# B&R Automation Studio project perfxxl (part 9)

#### flowcontrol.c
```c
#ifdef _DEFAULT_INCLUDES
	#include <AsDefault.h>
#endif
/*************************************************************************************************
 Flow control

 - checking Flow control sensor

*************************************************************************************************/

#include "egmglob_var.h"

BOOL				Pulse_1s,Overflow;
TON_10ms_typ		PulseTimer1;

_LOCAL	BOOL		CounterReset;

_LOCAL INT			DevCircFlowInv,PrewashFlowInv,RinseFlowInv,
					GumFlowInv, ReplFlowInv, TopUpFlowInv;

void FlowControl(FlowCount_type *FC,BOOL In, INT MinFreq)
{
	void NoFlow(void)
	{
		FC->LastCV = 0;
		FC->Flowing = FALSE;
		FC->EdgeCounter.RESET = TRUE;

		FC->LitersPerHour = 0;
		FC->LitersPerMinute = 0;
		FC->Frequency = 0;
		FC->OverflowCounter = 0;
	}

	if (Pulse_1s)
	{
		/*
		 * Sonderfall: wenn genau vor einem Zyklus ein Overflow stattfand
		 * dann ist aktueller Zählerstand = letzter Zählerstand = 0
		 * in dem Fall soll kein Reset erfolgen, sondern eine
		 * weitere Sekunde gewartet werden
		 */
		if( !Overflow )
		{
			if(FC->EdgeCounter.CV > FC->LastCV)
			{
				FC->Frequency = (FC->EdgeCounter.CV - FC->LastCV);
				FC->LastCV = FC->EdgeCounter.CV;
				if( FC->Frequency >= MinFreq )
				{
					FC->Flowing = TRUE;
					FC->LitersPerHour = (FC->Frequency / (REAL)FC->PulsesPerLiter)*3600.0;
					FC->LitersPerMinute = (FC->Frequency / (REAL)FC->PulsesPerLiter)*60.0;
				}
				else
					NoFlow();
			}
			else /* counter value has not been increased since 1 sec.: no flow */
				NoFlow();
		} /* if(!Overflow) */
		Overflow = FALSE;
	} /* if(Pulse_1s) */

/* reset value from somewhere else */
	if(FC->ResetMlFlown)
	{
		FC->ResetMlFlown = 0;
		FC->EdgeCounter.RESET = TRUE;
		FC->MlFlown = 0;
		FC->LastCV = 0;
		FC->OverflowCounter = 0;
	}

	if(CounterReset)
	{
		NoFlow();
		FC->MlFlown = 0;
	}

	/* counter overflow at 30000 */
	if(FC->EdgeCounter.CV >= 30000)
	{
		FC->EdgeCounter.RESET = TRUE;
		FC->LastCV = 0;
		FC->OverflowCounter++;
		Overflow = TRUE;
	}
	FC->EdgeCounter.CU = In;
	CTU(&(FC->EdgeCounter));
	FC->EdgeCounter.RESET = FALSE;

	if( FC->EdgeCounter.CV != 0 )
		FC->MlFlown = 1000.0 *
					( ((30000.0 * FC->OverflowCounter) + FC->EdgeCounter.CV)
					    / (REAL)FC->PulsesPerLiter
					 );
}

void InitFlowControl(FlowCount_type *FC)
{
	FC->EdgeCounter.CU = 0;
	FC->EdgeCounter.RESET = 1;
	FC->EdgeCounter.PV = 0;
	FC->OverflowCounter = 0;
	FC->LastCV = 0;
	FC->MlFlown = 0;
	FC->ResetMlFlown = 0;
}

_INIT void init(void)
{
	InitFlowControl(&GumFC);
	InitFlowControl(&ReplFC);
	InitFlowControl(&TopUpFC);

	PulseTimer1.IN = 0;
	PulseTimer1.PT = 100;
}

_CYCLIC void cyclic(void)
{
	DevCircFlowInv = !DevCircFlowInput;
	PrewashFlowInv = !PrewashFlowInput;
	RinseFlowInv = !RinseFlowInput;
	GumFlowInv = !GumFC.Flowing;
	ReplFlowInv = !ReplFC.Flowing;
	TopUpFlowInv = !TopUpFC.Flowing;

	PulseTimer1.IN = 1;
	if(PulseTimer1.Q)
		PulseTimer1.IN = 0;
	TON_10ms(&PulseTimer1);
	Pulse_1s = PulseTimer1.Q;

	if(    (EGMGlobalParam.GumPulsesPerLiter < 500)
		|| (EGMGlobalParam.GumPulsesPerLiter > 5000) )
		EGMGlobalParam.GumPulsesPerLiter = 1200;

	if(    (EGMGlobalParam.ReplenisherPulsesPerLiter < 500)
		|| (EGMGlobalParam.ReplenisherPulsesPerLiter > 5000) )
		EGMGlobalParam.ReplenisherPulsesPerLiter = 1200;

	if(    (EGMGlobalParam.DeveloperPulsesPerLiter < 500)
		|| (EGMGlobalParam.DeveloperPulsesPerLiter > 5000) )
		EGMGlobalParam.DeveloperPulsesPerLiter = 1200;

	GumFC.PulsesPerLiter = EGMGlobalParam.GumPulsesPerLiter;
	ReplFC.PulsesPerLiter = EGMGlobalParam.ReplenisherPulsesPerLiter;
	TopUpFC.PulsesPerLiter = EGMGlobalParam.DeveloperPulsesPerLiter;

	FlowControl(&GumFC,GumFlowInput,2);
	FlowControl(&ReplFC,ReplFlowInput,9);
	FlowControl(&TopUpFC,TopUpFlowInput,9);

}
```

### Program Logical/Processor/lccount (ANSIC, version 0.00.0)

#### lccount.c
```c
#ifdef _DEFAULT_INCLUDES
	#include <AsDefault.h>
#endif
/******************************************************************************************/
/*	LCCount aufrufen (Zeitbasis für Regler)*/
/**/
/******************************************************************************************/

#include "EGMglob_var.h"
#include <loopcont.h>

#define MM_PER_PULSE (251.0/17.0)

R_TRIGtyp	RPMSignalEdgeR;
/*timer für die Messung der Periodendauer des Antriebs-Taktes*/
REAL	tmpval,tmpval2,PeriodTime; /* in sec */

CTUtyp	PlateLengthCounter;

/*timer für die Messung der Periodendauer des Antriebs-Taktes*/
TON_typ	PeriodTimeRPM;
/*timer für die Messung der Verzögerung Plattenvorderkante->nächster Takt*/
TON_10ms_typ	PlateStartToRPMDelay;
/*timer für die Messung der Verzögerung Plattenhinterkante->nächster Takt*/
TON_10ms_typ	PlateEndToRPMDelay;
/*Var zum Speichern der gemessenen Zeiten*/
UDINT	StartDelay,EndDelay;

R_TRIGtyp	InputSensorEdgeR;
F_TRIGtyp	InputSensorEdgeF;
BOOL	 EnablePulseCounter;

_GLOBAL REAL PlateLength;
/* zum Entprellen des Eingangssensors*/
TON_10ms_typ	InputSensorOnDelay;
TOF_10ms_typ	InputSensorOffDelay;
_LOCAL REAL TEST;

/* ohne Mittelwertbildung */
void MeasureCurrentSpeed(void)
{

	RPMSignalEdgeR.CLK = RPMCheck;
	R_TRIG(&RPMSignalEdgeR);
/* steigende Flanke und timer ist gestartet: Zeit nehmen und stoppen*/
	if(RPMSignalEdgeR.Q )
	{
/* 2.02: Messung per Timer statt Zykluszähler */
		PeriodTime = PeriodTimeRPM.ET * 0.001; /* timer Wert 1 ms */
		PeriodTimeRPM.IN = FALSE;
	}
	else
		PeriodTimeRPM.IN = TRUE;
	PeriodTimeRPM.PT = 10000;
/* wenn 10 sec lang kein Takt, dann ist die Periodendauer 0 */
	if(PeriodTimeRPM.Q)
		PeriodTime = 0;

 	TON(&PeriodTimeRPM);
/* ENDE Periodendauer des Taktes messen*/
/*-------------------------------------------------------------------------------------------*/

/*-------------------------------------------------------------------------------------------*/
/* START Geschwindigkeit und Plattenlänge errechnen*/
/* Periodendauer ist gegen 0: Antrieb läuft nicht*/
/* Abfrage wichtig, da durch PeriodTime geteilt wird !!*/
	if (PeriodTime < 0.05)/* kürzer als 50 ms : ungültig, wäre 12 m/min*/
	{
		EGMGlobalParam.CurrentPlateSpeed = 0;
	}
	else
	{
/* 251mm/U / 17Takte/U =14.76 mm/Takt steht in MM_PER_PULSE */
/*PeriodTime*0.01 weil Timerwert in 10ms */
/* *0.06 weil Speed in m/min, Ergebnis vorher ist in mm/s*/
/* gilt so nur, wenn die Speed konstant ist, um schwankungen zu erfassen müsste man integrieren*/

	 	EGMGlobalParam.CurrentPlateSpeed = (MM_PER_PULSE / (PeriodTime))*0.06;
		tmpval = EGMGlobalParam.CurrentPlateSpeed / EGMGlobalParam.MainMotorFactor;
		if (tmpval <= 32767.0)
			EGMMainMotor.RealRpm = (INT)tmpval;
		else
			EGMMainMotor.RealRpm = 32767;

	}
/* ENDE Geschwindigkeit und Plattenlänge errechnen*/
/*-------------------------------------------------------------------------------------------*/
}

void MeasurePlateLength(void)
{

/**********************************************************************************/
/* Plattenlänge ermitteln*/

/*
Strategie für erhöhte Genauigkeit:
	- kontinuierlich Periodendauer des Taktsignals vom Antrieb messen (jede 2. Periode)
	- Zeit vom Erkennen des Plattenanfangs bis zum nächsten Takt messen
	- Zeit vom Erkennen des Plattenendes bis zum nächsten Takt messen
	- aus den gezählten Takten und den gemessenen Zeiten die Plattenlänge
	  ermitteln
*/

/*Entprellen je 1 sec*/
	InputSensorOnDelay.PT = 100;
	InputSensorOffDelay.PT = 100;
	InputSensorOnDelay.IN = InputSensor;
	InputSensorOffDelay.IN = InputSensor;
	TON_10ms(&InputSensorOnDelay);
	TOF_10ms(&InputSensorOffDelay);
	InputSensorEdgeR.CLK = InputSensorOnDelay.Q;
	InputSensorEdgeF.CLK = InputSensorOffDelay.Q;
	R_TRIG(&InputSensorEdgeR);
	F_TRIG(&InputSensorEdgeF);

/*-------------------------------------------------------------------------------------------*/
/* START Messung Verzögerung Plattenvorderkante->nächster Takt*/
/*mit steigender Flanke des Sensors Zeitmessung starten*/
	PlateStartToRPMDelay.PT = 60000;
	if (InputSensorEdgeR.Q && !PlateStartToRPMDelay.IN)
		PlateStartToRPMDelay.IN = 1;
/*bei der nächsten steigenden Flanke des Taktes die Zeit nehmen*/
/* || PlateStartToRPMDelay.Q nur für den Fall, dass der Antrieb steht o.ä.*/
	if (PlateStartToRPMDelay.IN && (RPMSignalEdgeR.Q || PlateStartToRPMDelay.Q ))
	{
		PlateStartToRPMDelay.IN = 0;
		StartDelay = PlateStartToRPMDelay.ET;
	}
	TON_10ms(&PlateStartToRPMDelay);
/* ENDE Messung Verzögerung Plattenvorderkante->nächster Takt*/
/*-------------------------------------------------------------------------------------------*/

/*-------------------------------------------------------------------------------------------*/
/* START Messung Verzögerung Plattenhinterkante->nächster Takt*/
/*mit steigender Flanke des Sensors Zeitmessung starten*/
	PlateEndToRPMDelay.PT = 60000;
	if (InputSensorEdgeF.Q && !PlateEndToRPMDelay.IN)
		PlateEndToRPMDelay.IN = 1;
/*bei der nächsten steigenden Flanke des Taktes die Zeit nehmen*/
/* || PlateEndToRPMDelay.Q nur für den Fall, dass der Antrieb steht o.ä.*/
	if (PlateEndToRPMDelay.IN && (RPMSignalEdgeR.Q || PlateEndToRPMDelay.Q ))
	{
		PlateEndToRPMDelay.IN = 0;
		EndDelay = PlateEndToRPMDelay.ET;
	}
	TON_10ms(&PlateEndToRPMDelay);
/* ENDE Messung Verzögerung Plattenhinterkante->nächster Takt*/
/*-------------------------------------------------------------------------------------------*/

/*-------------------------------------------------------------------------------------------*/
/* START Zählen der Takte, während Platte durchläuft*/
	CTU(&PlateLengthCounter);

/*bei fallender Flanke den Zähler auswerten*/
	if(InputSensorEdgeF.Q)
	{
/* nicht durch 0 teilen... */
		if(PeriodTime < 0.05)
			tmpval2 = PlateLengthCounter.CV;
		else
			tmpval2 = PlateLengthCounter.CV+ ((REAL)StartDelay)/(PeriodTime*100.0) - ((REAL)EndDelay)/(PeriodTime*100.0);
		PlateLength = tmpval2 * MM_PER_PULSE;
		if (PlateLength < 0.0) PlateLength = 0.0;
		if (PlateLength > 3000.0) PlateLength = 0.0;
		EnablePulseCounter = 0;
	}
/* mit Einlaufstart den Pulszähler enablen*/
	if(InputSensorEdgeR.Q)
	{
		EnablePulseCounter = 1;
	}
	if (EnablePulseCounter)
	{
		PlateLengthCounter.CU = RPMCheck;
	}
/*zur Sicherheit den Pulscounter disablen, wenn keine Platte im Einlaufbereich ist*/
	if ( !InputSensorOnDelay.Q && !InputSensorOffDelay.Q)
		EnablePulseCounter = 0;

/*bei Start einer Platte Zähler resetten, Takte zählen*/
	PlateLengthCounter.RESET = InputSensorEdgeR.Q;

/* ENDE Zählen der Takte, während Platte durchläuft*/
/*-------------------------------------------------------------------------------------------*/
}

_INIT void init(void)
{
	PlateLength = 0;
/*	PeriodTimeCounter = 0;*/
	PeriodTime = 0;
	PeriodTimeRPM.IN = FALSE;
}

_CYCLIC void cyk(void)
{
	LCCounter(&LCCountVar);
	MeasureCurrentSpeed();
	MeasurePlateLength();
}
```

- egmglob_var.h (reference to Logical/GlobalIncludes/egmglob_var.h)

### Program Logical/Processor/egmio (ANSIC, version 0.00.0)

#### egm_in_out.c
```c
#ifdef _DEFAULT_INCLUDES
	#include <AsDefault.h>
#endif
#include "glob_var.h"
#include "egmglob_var.h"

#define OUTMODULES (3)
#define OUTPUTSPERMODULE (12)

_LOCAL    BOOL                EGMModule1Out[12];
_LOCAL    BOOL                EGMModule2Out[12];
_LOCAL    BOOL                EGMModule3Out[12];
_LOCAL    BOOL                EGMModule1In[12];
_LOCAL    BOOL                EGMModule2In[12];

static BOOL dummy;

_INIT void i(void)
{
	MachineType = BLUEFIN_LOWCHEM;
/*	MachineType = BLUEFIN_XS;*/
}

_CYCLIC void c(void)
{

/*
Maschinenlänge in m
	Standard Bluefin 2.80
	XS Bluefin		 2.70
	LowChem Bluefin  2.05
 */

	if(MachineType == BLUEFIN_XS)
	{
		MACHINELENGTH = 2.70;
	/* XS Output */
		EGMModule1Out[0] = Horn;
		EGMModule1Out[1] = LightGreen;
		EGMModule1Out[2] = LightYellow;
		EGMModule1Out[3] = LightRed;
		EGMModule1Out[4] = EGMMainMotor.Enable;
		EGMModule1Out[5] = EGMBrushMotor.Enable;
		EGMModule1Out[6] = Ready;
		EGMModule1Out[7] = NoError;
		EGMModule1Out[8] = ActivateControlVoltage;
		EGMModule1Out[9] = EGMPrewash.Valve;
		EGMModule1Out[10] = EGMRinse.Valve;
		EGMModule1Out[11] = EGMGum.RinseValve;

		EGMModule2Out[0] = HeatingON[0];
		EGMModule2Out[1] = HeatingON[1];
		EGMModule2Out[2] = HeatingON[2];
		EGMModule2Out[3] = HeatingON[3];
		EGMModule2Out[4] = EGMDeveloperTank.HeatingOn;
		EGMModule2Out[5] = EGMGum.Valve;
		EGMModule2Out[6] = EGMDeveloperTank.CoolingOn;
		EGMModule2Out[7] = FALSE;
		EGMModule2Out[8] = FALSE;
		EGMModule2Out[9] = FALSE;
		EGMModule2Out[10] = FALSE;
		EGMModule2Out[11] = FALSE;

		EGMModule3Out[0] = EGMPrewash.Pump;
		EGMModule3Out[1] = EGMRinse.Pump;
		EGMModule3Out[2] = EGMPreheat.FansOn;
		EGMModule3Out[3] = Drying;
		if(EGMGlobalParam.PROV_KitInstalled)
			EGMModule3Out[4] = Out_DevCanister_Circulation;
		else
			EGMModule3Out[4] = EGMDeveloperTank.RegenerationPump;
		EGMModule3Out[5] = EGMGum.Pump;
		EGMModule3Out[6] = EGMDeveloperTank.CirculationPump;
		if(EGMGlobalParam.PROV_KitInstalled)
			EGMModule3Out[7] = Out_DevCanister_Replenish;
		else
			EGMModule3Out[7] = EGMDeveloperTank.Refill;
		EGMModule3Out[8] = FALSE;
		EGMModule3Out[9] = FALSE;
		EGMModule3Out[10] = FALSE;
		EGMModule3Out[11] = FALSE;

	/* XS Input */
		ControlVoltageOk 			= EGMModule1In[0];
		RPMCheck 					= EGMModule1In[1];
		InputSensor 				= EGMModule1In[2];
		EGMPrewash.TankFull 		= EGMModule1In[3];
		EGMRinse.TankFull 			= EGMModule1In[4];
		EGMGum.TankFull				= EGMModule1In[5];
		EGMDeveloperTank.TankFull	= EGMModule1In[6];
/*                                                 7 s.u.ProV */
		OutputSensor				= EGMModule1In[8];
		ServiceKey					= EGMModule1In[9];
		VCP_OK						= EGMModule1In[10];
		if(EGMGlobalParam.PROV_KitInstalled)
		{
			In_DevCanister_Full			= EGMModule1In[7];
			In_DevCanister_Empty		= EGMModule1In[11];
		}
		else
		{
			dummy						= EGMModule1In[7];
			dummy						= EGMModule1In[11];
		}

		GumFlowInput	 			= EGMModule2In[0];
		ReplFlowInput	 			= EGMModule2In[1];
		TopUpFlowInput	 			= EGMModule2In[2];
		DevCircFlowInput 			= EGMModule2In[3];
		PrewashFlowInput	 		= EGMModule2In[4];
		RinseFlowInput	 			= EGMModule2In[5];
/*		In_WasteTankNearlyFull		= EGMModule2In[6];
		In_WasteTankFull 			= EGMModule2In[7];*/
		dummy						= EGMModule2In[8];
		dummy						= EGMModule2In[9];
		dummy						= EGMModule2In[10];
		dummy						= EGMModule2In[11];
	}
	else
	if(MachineType == BLUEFIN_LOWCHEM)
	{
		EGMGlobalParam.PROV_KitInstalled = FALSE;
		MACHINELENGTH = 2.05;
	/* LowChem Output */
		EGMModule1Out[0] = Horn;
		EGMModule1Out[1] = LightGreen;
		EGMModule1Out[2] = LightYellow;
		EGMModule1Out[3] = LightRed;
		EGMModule1Out[4] = EGMMainMotor.Enable;
		EGMModule1Out[5] = EGMBrushMotor.Enable;
		EGMModule1Out[6] = ActivateControlVoltage;
		EGMModule1Out[7] = FALSE;
		EGMModule1Out[8] = FALSE;
		EGMModule1Out[9] = FALSE;
		EGMModule1Out[10] = EGMGum.Valve;
		EGMModule1Out[11] = EGMGum.RinseValve;

		EGMModule2Out[0] = HeatingON[0];
		EGMModule2Out[1] = HeatingON[1];
		EGMModule2Out[2] = EGMDeveloperTank.HeatingOn;
		EGMModule2Out[3] = FALSE;
		EGMModule2Out[4] = FALSE;
		EGMModule2Out[5] = FALSE;
		EGMModule2Out[6] = EGMDeveloperTank.CoolingOn;
		EGMModule2Out[7] = FALSE;
		EGMModule2Out[8] = FALSE;
		EGMModule2Out[9] = FALSE;
		EGMModule2Out[10] = FALSE;
		EGMModule2Out[11] = FALSE;

		EGMModule3Out[0] = EGMPrewash.Pump;
		EGMModule3Out[1] = EGMRinse.Pump;
		EGMModule3Out[2] = EGMPreheat.FansOn;
		EGMModule3Out[3] = Drying;
		EGMModule3Out[4] = EGMDeveloperTank.RegenerationPump;
		EGMModule3Out[5] = EGMGum.Pump;
		EGMModule3Out[6] = EGMDeveloperTank.CirculationPump;
		EGMModule3Out[7] = EGMDeveloperTank.Refill;
		EGMModule3Out[8] = FALSE;
		EGMModule3Out[9] = FALSE;
		EGMModule3Out[10] = Ready;
		EGMModule3Out[11] = NoError;

	/* LowChem Input */
		ControlVoltageOk 			= EGMModule1In[0];
		RPMCheck 					= EGMModule1In[1];
		InputSensor 				= EGMModule1In[2];
		DevCircFlowInput	 		= EGMModule1In[3];
		TopUpFlowInput	 			= EGMModule1In[4];
		EGMGum.TankFull				= EGMModule1In[5];
		EGMDeveloperTank.TankFull	= EGMModule1In[6];
		GumFlowInput				= EGMModule1In[7];
		OutputSensor				= EGMModule1In[8];
		ServiceKey					= EGMModule1In[9];
		VCP_OK						= EGMModule1In[10];
		dummy						= EGMModule1In[11];

		dummy						= EGMModule2In[0];
		ReplFlowInput	 			= EGMModule2In[1];
		dummy						= EGMModule2In[2];
		dummy						= EGMModule2In[3];
		dummy						= EGMModule2In[4];
		dummy						= EGMModule2In[5];
		dummy						= EGMModule2In[6];
		dummy						= EGMModule2In[7];
		dummy						= EGMModule2In[8];
		dummy						= EGMModule2In[9];
		dummy						= EGMModule2In[10];
		dummy						= EGMModule2In[11];
	}
}
```

- egmglob_var.h (reference to Logical/GlobalIncludes/egmglob_var.h)

### Program Logical/Processor/motors (ANSIC, version 0.00.0)

#### motors.c
```c
#ifdef _DEFAULT_INCLUDES
	#include <AsDefault.h>
#endif
/*************************************************************************************************
 Handling of Motors
 - Main Motor (Propulsion of plate)
 - Brush Motor

*************************************************************************************************/

#include "glob_var.h"
#include "egmglob_var.h"
#include <math.h>

TP_10ms_typ		RPMCheckTimer;
F_TRIGtyp 			RPMCheckEdge;
CTUtyp	RPMEdgeCounter;
_LOCAL	UINT	CounterValue;
TON_10ms_typ		BrushMotorOnTimer1,BrushMotorOnTimer2;
TON_10ms_typ		RPMSignalCheckTimer,RPMDeviationTimer;
/* Input delay timer for ControlVoltage signal */
TON_10ms_typ		ControlVoltageOkDelay;

REAL	tmpval;

TON_10ms_typ	PulseTimer1;
BOOL	Pulse_1s;
_LOCAL REAL MainMotorFactorFeet;

_INIT void init()
{
	CounterValue = 0;
	EGMMainMotor.RatedRpm = 0;
	EGMMainMotor.RealRpm = 0;
	EGMMainMotor.Auto = 0;
	EGMMainMotor.Enable = 0;

	EGMBrushMotor.RatedRpm = 0;
	EGMBrushMotor.RealRpm = 0;
	EGMBrushMotor.Auto = 0;
	EGMBrushMotor.Enable = 0;

	BrushMotorOnTimer1.IN = 0;
	BrushMotorOnTimer2.IN = 0;

	PulseTimer1.IN = 0;
	PulseTimer1.PT = 100; /* 1 sec */

}

_CYCLIC void cyclic()
{
	PulseTimer1.IN = 1;
	if(PulseTimer1.Q)
		PulseTimer1.IN = 0;
	TON_10ms(&PulseTimer1);
	Pulse_1s = PulseTimer1.Q;

/* Skalierungsfaktor muss in VC Einheitengruppe "Vorschub" identisch sein !! */
/*	EGMGlobalParam.MainMotorFactor = 9.30814539017914E-05;*/
	MainMotorFactorFeet = EGMGlobalParam.MainMotorFactor / 0.3048;
/* das gleiche für Bürstenmotor */
/*  "Alter" Motortyp*/
/*	EGMGlobalParam.BrushFactor = 180.0/32767.0;*/
/*  "Neuer" Motortyp Siemens*/
/*	EGMGlobalParam.BrushFactor = 230.0/32767.0;*/

/* safety:
 * 	Not a number or out of reasonable range ->set default*/
	if( isnan(EGMGlobalParam.BrushFactor)
	 || (EGMGlobalParam.BrushFactor > 0.02)  /* > ca 655 rpm */
	 || (EGMGlobalParam.BrushFactor < 0.001) /* < ca 32.7 rpm */
	  )
		EGMGlobalParam.BrushFactor = 230.0/32767.0;

/*Main Motor*/
/* safety:
 * 	Not a number or out of reasonable range ->set default*/
	if( isnan(EGMGlobalParam.MainMotorFactor)
	 || (EGMGlobalParam.MainMotorFactor > (10.0/32767.0))
	 || (EGMGlobalParam.MainMotorFactor < 1.0/32767.0)
	  )
		EGMGlobalParam.MainMotorFactor = 3.0/32767.0;

	EGMMainMotor.Manual = !EGMMainMotor.Auto;

/**
Prüfen, ob überhaupt Signale vom Taktsensor kommen:
Wenn Sollwert > 0,2 m/min, dann muss der Countervalue > 0 sein
*/
	RPMSignalCheckTimer.IN = ((CounterValue == 0) && ((EGMMainMotor.RatedRpm * EGMGlobalParam.MainMotorFactor)> 0.2 ));
	RPMSignalCheckTimer.PT = 1000; /* 10 sec */
	TON_10ms(&RPMSignalCheckTimer);
	EGM_AlarmBitField[1] = RPMSignalCheckTimer.Q;

	RPMDeviationTimer.PT = 1000;
	RPMDeviationTimer.IN = ((fabs((EGMGlobalParam.MainMotorFactor*EGMMainMotor.RatedRpm) - EGMGlobalParam.CurrentPlateSpeed)) > 0.5)
							&& !EGM_AlarmBitField[1] && EGMMainMotor.Enable && !CurrentState==S_OFF && ControlVoltageOk;
	TON_10ms(&RPMDeviationTimer);
	EGM_AlarmBitField[27] = RPMDeviationTimer.Q;

/* Messung der Speed über Taktgeber*/
	RPMEdgeCounter.CU = RPMCheck;
	RPMEdgeCounter.PV = 32000; /*soll nicht erreicht werden*/

	CTU(&RPMEdgeCounter);
	RPMEdgeCounter.RESET = 0;

	TP_10ms(&RPMCheckTimer);

	RPMCheckTimer.IN = Pulse_1s;
	RPMCheckTimer.PT = 1000; /*10 sec Messen*/

/*fallende Flanke des Pulstimers auswerten*/
	RPMCheckEdge.CLK	= RPMCheckTimer.Q;
	F_TRIG(&RPMCheckEdge);

	if (RPMCheckEdge.Q)
	{
		CounterValue = RPMEdgeCounter.CV;
		RPMEdgeCounter.RESET = 1;
	}

/*im Automatik-Modus die Auto-Drehzahl übernehmen*/
/*-> im Hand Modus kann man dann die RatedRpm direkt verändern*/
/*Spannung muß schon 5 sec lang anliegen, sonst erkennt FU das Signal nicht zuverlässig*/
	ControlVoltageOkDelay.IN = ControlVoltageOk;
	ControlVoltageOkDelay.PT = 500;
	TON_10ms(&ControlVoltageOkDelay);
	if (EGMMainMotor.Auto && ControlVoltageOkDelay.Q)
	{
		EGMMainMotor.Enable = 1;	/* Freigabe Ausgang an FU */
		EGMMainMotor.RatedRpm = EGMMainMotor.AutoRatedRpm;	/* Drehzahl Ausgang an FU */
	}

	if (!ControlVoltageOk)
	{
		EGMMainMotor.Enable = 0;	/* Freigabe Ausgang an FU */
		EGMMainMotor.Auto = 0;
	}

/*************************************************************************************************/

/*Brush Motor*/
	EGMBrushMotor.Manual = !EGMBrushMotor.Auto;
/*keine Messung: Ist = Soll*/
	EGMBrushMotor.RealRpm = EGMBrushMotor.RatedRpm;
/*im Automatik-Modus die Auto-Drehzahl übernehmen*/
/*-> im Hand Modus kann man dann die RatedRpm direkt verändern*/
	if (EGMBrushMotor.Auto && ControlVoltageOkDelay.Q)
	{
		EGMBrushMotor.Enable = 1;	/* Freigabe Ausgang an FU */
/*
		if (BrushMotorOnTimer2.IN )
			EGMBrushMotor.RatedRpm = 150.0 / EGMGlobalParam.BrushFactor;
		else
 */
			EGMBrushMotor.RatedRpm = EGMBrushMotor.AutoRatedRpm;	/* Drehzahl Ausgang an FU */
	}

	if (!ControlVoltageOk)
	{
		EGMBrushMotor.Enable = 0;	/* Freigabe Ausgang an FU */
		EGMBrushMotor.Auto = 0;
	}

	if (EGMBrushMotor.Auto && (EGMBrushMotor.RatedRpm < 100.0/EGMGlobalParam.BrushFactor) )
	{
		BrushMotorOnTimer1.IN = 1;
	}
	else
		BrushMotorOnTimer1.IN = 0;

	BrushMotorOnTimer1.PT = 9000; /* alle 1,5 min*/
	TON_10ms(&BrushMotorOnTimer1);

	BrushMotorOnTimer2.PT = 2000; /* 20 sec*/
	TON_10ms(&BrushMotorOnTimer2);

/* nach Zeit die Bürsten hochdrehen*/
	if (BrushMotorOnTimer1.Q  )
	{
		BrushMotorOnTimer2.IN = 1;
	}

	if (BrushMotorOnTimer2.Q)
	{
		BrushMotorOnTimer2.IN = 0;
	}
}
```

### Program Logical/Processor/preheat (ANSIC, version 0.00.0)

#### preheat.c
```c
#ifdef _DEFAULT_INCLUDES
	#include <AsDefault.h>
#endif
/*************************************************************************************************
 Handling of Preheat

 - Heating, Temperature Measurement

*************************************************************************************************/

#include "EGMglob_var.h"

extern void PreheatPID(void);
extern void PreheatPID_DefaultParam(void);

int i;
_GLOBAL BOOL	HeatingON[4];
_INIT void init()
{

	PreheatPID_DefaultParam();
}

_CYCLIC void cyclic()
{

	PreheatPID();
	return;
}
```

#### preheat_pid.c
```c
#ifdef _DEFAULT_INCLUDES
	#include <AsDefault.h>
#endif
/*****************************************************************************************/
/*	Preheat regelung mit LoopCont Library*/
/*	wird aus EGMPreheat.c aufgerufen*/
/*****************************************************************************************/

/*
#define TESTCURVE
*/
/**/
#undef TESTCURVE
/**/

#include <math.h>
#include "EGMglob_var.h"
#include "auxfunc.h"

/*für Sollwertnachführung*/
#define NUMBER_OF_POINTS		720 /*2h lang alle 10 sec ein wert*/
#define NUMBER_OF_SECONDS	7200 /*2h */
/*für Stabilitätscheck*/
#define NUMBER_OF_RANGECHECK_SECONDS	30
#define OVERHEATTEMP 500	/* 50 °C über der Solltemp.*/

_GLOBAL SINT IOConfiguration	_VAR_RETAIN;

_LOCAL	LCPWM_DMod_typ		LCPWM_DMod_var[MAX_NUMBER_OF_CONTROLLERS];
_LOCAL	LCPIDpara_typ			LCPIDpara_var[MAX_NUMBER_OF_CONTROLLERS];
_LOCAL	LCPID_typ				LCPID_var[MAX_NUMBER_OF_CONTROLLERS];
_LOCAL	LCPIDAutoTune_typ		LCPIDAutoTune_var[MAX_NUMBER_OF_CONTROLLERS];
_LOCAL	LCCurveByPoints_typ	LCCurveByPoints_var,LCCurveByPoints_var2;

/*Feld für Kurve der Sollwertnachführung*/
/* e-Funktion*/
_LOCAL lcCurveByPoints_TabEntry_type   CurveByPoints_Table[NUMBER_OF_POINTS];
/* Korrekturen der e-Funktion*/
_LOCAL lcCurveByPoints_TabEntry_type   CurveByPoints_Table2[15];

_LOCAL	BOOL 	StartAutoTune;
_LOCAL	BOOL	TriggerLogging,TriggerLoggingOld;
TON_10ms_typ	Pulse,PulseTimer1;
TON_10ms_typ		HeatingFailureTimer[MAX_NUMBER_OF_CONTROLLERS];

int i;
_GLOBAL int	Values[350];
_GLOBAL int	AmbientValues[350];

int	RangeCheckArray[MAX_NUMBER_OF_CONTROLLERS][NUMBER_OF_RANGECHECK_SECONDS];
int ValueCount,RangeCheckCount,SPTrackCount;
BOOL flag[MAX_NUMBER_OF_CONTROLLERS];
_GLOBAL BOOL RedrawCurve,PreheatParamEnter;
_GLOBAL	UINT	SamplingTime;
BOOL	StopSPTracking;
BOOL	Overheated;
INT LastTemp[MAX_NUMBER_OF_CONTROLLERS];

R_TRIGtyp	InputSensorEdgeR;
F_TRIGtyp	InputSensorEdgeF;
TON_10ms_typ	InputSensorOnDelay;
TOF_10ms_typ	InputSensorOffDelay;
int	PlateInputCounter;
int TempCorrectionValue;
int SecWithoutPlate;

/* depending on Bluefin-Variant: Standard or 1250 */
_LOCAL    INT                 ActualNumberOfControllers;

void Preset_CorrCurve(void)
{
	int i;
	REAL k;

/*e-Funktion für Startup erzeugen*/
	for (i=0;i<NUMBER_OF_POINTS;i++)
	{
		CurveByPoints_Table[i].x = i*(NUMBER_OF_SECONDS / NUMBER_OF_POINTS) ;

		k = -((float)NUMBER_OF_SECONDS / (float) NUMBER_OF_POINTS)  / (60.0* EGMPreheatParam.SetPointCorrTMin);
		CurveByPoints_Table[i].y = EGMPreheatParam.SetPointCorrMax * exp(k*i);
	}

/*initialisieren der Korrekturkurve für die e-Funktion*/
	for (i=0;i<15;i++)
	{
		CurveByPoints_Table2[i].x = 0;
		CurveByPoints_Table2[i].y = 0;
	}
/*und mit Stützpunkten füllen*/
/* 1 */
	CurveByPoints_Table2[0].x = 0;
	CurveByPoints_Table2[0].y = 0;
/* 2 */
	CurveByPoints_Table2[1].x = 180;
	CurveByPoints_Table2[1].y = -50;
/* 3 */
	CurveByPoints_Table2[2].x = 300;
	CurveByPoints_Table2[2].y = -80;
/* 4 */
	CurveByPoints_Table2[3].x = 540;
	CurveByPoints_Table2[3].y = -90;
/* 5 */
	CurveByPoints_Table2[4].x = 840;
	CurveByPoints_Table2[4].y = -110;
/* 6 */
	CurveByPoints_Table2[5].x = 1200;
	CurveByPoints_Table2[5].y = -80;
/* 7 */
	CurveByPoints_Table2[6].x = 1740;
	CurveByPoints_Table2[6].y = -60;
/* 8 */
	CurveByPoints_Table2[7].x = 2700;
	CurveByPoints_Table2[7].y = -30;
/* 9 */
	CurveByPoints_Table2[8].x = 3480;
	CurveByPoints_Table2[8].y = -10;
/* 10 */
	CurveByPoints_Table2[9].x = 3660;
	CurveByPoints_Table2[9].y = 0;
/* 11 */
	CurveByPoints_Table2[10].x = 4860;
	CurveByPoints_Table2[10].y = 0;
/* 12 */
	CurveByPoints_Table2[11].x = 5400;
	CurveByPoints_Table2[11].y = 10;
/* 13 */
	CurveByPoints_Table2[12].x = 6000;
	CurveByPoints_Table2[12].y = 25;
/* 14 */
	CurveByPoints_Table2[13].x = 6660;
	CurveByPoints_Table2[13].y = 19;

}

void PreheatPID_DefaultParam(void)
{
	int j;

/* depending on IO config we have 2 or 4 Controllers running*/
	switch (IOConfiguration)
	{
		case 1 /* Standard Bluefin */:
		{
			ActualNumberOfControllers = 2;
			break;
		}
		case 2 /* Bluefin 1250 */:
		{
			ActualNumberOfControllers = 4;
			break;
		}
		default:
		{
			ActualNumberOfControllers = 2;
			break;
		}
	}
	PreheatParamEnter = 0;
	StopSPTracking = 0;
	SamplingTime = 100;
	SPTrackCount = 0;
	PulseTimer1.PT = 100;

	LCCurveByPoints_var.ptr_table = &CurveByPoints_Table[0];
	LCCurveByPoints_var.NoOfPoints = NUMBER_OF_POINTS;

	LCCurveByPoints_var2.ptr_table = &CurveByPoints_Table2[0];
	LCCurveByPoints_var2.NoOfPoints = 14;

	Preset_CorrCurve();

	for (i=0;i<ActualNumberOfControllers;i++)
	{
		LCPWM_DMod_var[i].tminpuls			= 10;  /* 10 ms kürzester Puls bzw pause*/
		LCPWM_DMod_var[i].tperiod			= 200;  /*Periodendauer 0,2 sec*/
		LCPWM_DMod_var[i].enable			= 1;
		LCPWM_DMod_var[i].max_value	= 100;
		LCPWM_DMod_var[i].min_value		= 0;

/*Sollwertabschwächung (1=AUS)*/
		LCPIDpara_var[i].Kw						= 1;
/*windup Dämpfung: 0=AUS*/
		LCPIDpara_var[i].Kfbk						= 0;
		LCPIDpara_var[i].enable					= 1;
		LCPIDpara_var[i].Y_max				= 100;
		LCPIDpara_var[i].Y_min					= 0;
		LCPIDpara_var[i].dY_max				= 0; /* 0= keine Rampe*/
	/*
	Rückführmodus der Stellgröße
	LCPID_FBK_MODE_INTERN: intern
	LCPID_FBK_MODE_EXTERN: extern für Ablöseregelung
	LCPID_FBK_MODE_EXT_SELECTOR: extern für Selektorregelung. In diesem Modus wird der I-Anteil des momentan nicht selektierten Reglers (Y_fbk ? Y) nach der
	Formel Yi = Y_fbk – Yp – Yd – A dem Eingang Y_fbk nachgeführt.
	*/
		LCPIDpara_var[i].fbk_mode				= LCPID_FBK_MODE_INTERN;
	/*
	Differenziermodus
	LCPID_D_MODE_X: nur -X (Istwert)
	LCPID_D_MODE_E: e (Regelabweichung, wie bei einem Standard- PID- Regler )
	*/
		LCPIDpara_var[i].d_mode				= LCPID_D_MODE_X;
	/*
	Rechenmodus:
	LCPID_CALC_MODE_EXACT: Genau (Alle Berechnungen erfolgen in Double Float - keine Rundungsfehler, auf SG3-Zentraleinheiten lange Rechenzeiten).
	LCPID_CALC_MODE_FAST: Schnell (Alle Berechnungen erfolgen in Integer - es kann zu geringfügigen Rundungsfehlern kommen, wird auch auf SG3-Zentraleinheiten sehr schnell gerechnet)
	*/
		LCPIDpara_var[i].calc_mode			= LCPID_CALC_MODE_EXACT;

/* Reglerbaustein LCPID*/
		LCPID_var[i].enable					= 1;
/*Stellgröße Handbetrieb */
		LCPID_var[i].Y_man					= 0;
	/*Aufschaltgröße*/
		LCPID_var[i].A							= 0;
	/*I-Anteil einfrieren*/
		LCPID_var[i].hold_I					= 0;

/* Autotune*/
		LCPIDAutoTune_var[i].enable				= 1;
		LCPIDAutoTune_var[i].Y_max				= 100;
		LCPIDAutoTune_var[i].Y_min				= 0;
		LCPIDAutoTune_var[i].P_manualAdjust		= 0;
		LCPIDAutoTune_var[i].I_manualAdjust		= 0;
		LCPIDAutoTune_var[i].D_manualAdjust		= 0;

		EGMPreheat.Auto[i] = 0;

		TriggerLogging = 0;
		for(j=0;j<NUMBER_OF_RANGECHECK_SECONDS;j++)
			RangeCheckArray[i][j] = 200;
	}
	RangeCheckCount = 0;
	i=0;
	ValueCount = 0;
	InputSensorOnDelay.IN = 0;
	InputSensorOffDelay.IN = 0;
	SecWithoutPlate = 0;
	TempCorrectionValue = 0;
	for(i=0;i<ActualNumberOfControllers;i++)
	{
		LastTemp[i] = 0;
		HeatingFailureTimer[i].IN = 0;
		HeatingFailureTimer[i].PT = 1000;
	}
}

/***********************************************************************
*                                                                      *
*                                                                      *
*     Sollwert pro Platte sukzessive erhöhen, nach Zeit ohne Platte    *
*     wieder verringern                                                *
*                                                                      *
*                                                                      *
***********************************************************************/
void SetpointCorrectionPerPlate(void)
{
/*Flankenerkennung Inputsensor */
	InputSensorEdgeR.CLK = InputSensorOnDelay.Q;
	InputSensorEdgeF.CLK = InputSensorOffDelay.Q;
	R_TRIG(&InputSensorEdgeR);
	F_TRIG(&InputSensorEdgeF);

	InputSensorOnDelay.PT = 100;
	InputSensorOffDelay.PT = 100;
/*Entprellen je 1 sec*/
	InputSensorOnDelay.IN = InputSensor;
	InputSensorOffDelay.IN = InputSensor;
	TON_10ms(&InputSensorOnDelay);
	TOF_10ms(&InputSensorOffDelay);

	if( InputSensor )
		SecWithoutPlate = 0;
	else
	if( PulseTimer1.Q ) /* Pulse every sec */
	{
		SecWithoutPlate++;
		if( (SecWithoutPlate % 60) == 0) /* every minute */
		{
			TempCorrectionValue += EGMPreheatParam.IncPerMinute;
			if( TempCorrectionValue > 0 )
				TempCorrectionValue = 0;
		}
	}

/* Platte läuft ein */
	if( InputSensorEdgeF.Q )
	{
		SecWithoutPlate = 0;	/* nur zur Sicherheit */
/* wenn Umgebunstemp. > Schwellwert*/
		if( EGMPreheat.AmbientTemp[0] > EGMPreheatParam.AmbientThreshold )
		{
			TempCorrectionValue -= EGMPreheatParam.DecPerPlate;
			if( abs(TempCorrectionValue) > abs(EGMPreheatParam.MaxInc) )
				TempCorrectionValue = EGMPreheatParam.MaxInc;
		}
	}

}

/***********************************************************************
*                                                                      *
*     PID Regler Funktionalität für beide Preheat Kreise               *
*                                                                      *
*                                                                      *
***********************************************************************/
void PreheatPID(void)
{
	int j;
	int k;
/*
	SetpointCorrectionPerPlate();
*/
	TempCorrectionValue = 0; /* rausnehmen, wenn Aufruf von SetpointCorrectionPerPlate
	                          * wieder einkommentiert wird !!
                              */

/* depending on IO config we have 2 or 4 Controllers running*/
	switch (IOConfiguration)
	{
		case 1 /* Standard Bluefin */:
		{
			ActualNumberOfControllers = 2;
			break;
		}
		case 2 /* Bluefin 1250 */:
		{
			ActualNumberOfControllers = 4;
			break;
		}
		default:
		{
			ActualNumberOfControllers = 2;
			break;
		}
	}

	for (j=0;j<ActualNumberOfControllers;j++)
		EGMPreheat.HeatingOn[j] = HeatingON[j];

/* Preheat enabled: Fans on as soon as Controlvoltage is on*/
	if( EGMPreheat.Enable )
		EGMPreheat.FansOn = ControlVoltageOk;
	else /* Preheat Off and Temp. in both Heatings < 100 °C
	      * or Emergency stop
	      * -> Fans OFF
	      */
	if( !ControlVoltageOk ||
	    (EGMPreheat.RealTemp[0] < 1000
	 &&  EGMPreheat.RealTemp[1] < 1000
	 && (LCPWM_DMod_var[0].x == 0)
	 && (LCPWM_DMod_var[1].x == 0))
	  )
		EGMPreheat.FansOn = 0;
	else	/* Preheat OFF, Controlvoltage ON, but both heatings >110 °C
	         * or one heating is ON -> Fans on
	         */
	if( ((EGMPreheat.RealTemp[0] > 1100) && ( EGMPreheat.RealTemp[1] > 1100 ))
	   || (LCPWM_DMod_var[0].x != 0)
	   || (LCPWM_DMod_var[1].x != 0)
	)
		EGMPreheat.FansOn = 1;

/**
Heizung defekt erkennen:
Ausgang 100% aber Temperatur steigt nicht
Erkennung für beide Heizkreise einzeln
**/
	for (i = 0;i<ActualNumberOfControllers;i++)
	{
		HeatingFailureTimer[i].IN = (LCPWM_DMod_var[i].x == 100) && !HeatingFailureTimer[i].Q;
		TON_10ms(&HeatingFailureTimer[i]);

		if( HeatingFailureTimer[i].Q )
		{
			/*
			 * 10 sec 100% Heating, but no rising temp. -> Alarm on
			*/
/* alarms for 1 and 2 are number 19 and 20*/
			if(i<2)
			{
				if( EGMPreheat.RealTemp[i] <= LastTemp[i]+10)
					EGM_AlarmBitField[19+i] = 1;
				else	/* Temp. did rise: Alarm off*/
					EGM_AlarmBitField[19+i] = 0;
			}
/* alarms for 3 and 4 are number 29 and 30*/
			else
			{
				if( EGMPreheat.RealTemp[i] <= LastTemp[i]+10)
					EGM_AlarmBitField[29+i] = 1;
				else	/* Temp. did rise: Alarm off*/
					EGM_AlarmBitField[29+i] = 0;
			}

			/* save current temp. for next check in 10 sec */
			LastTemp[i] = EGMPreheat.RealTemp[i];
		}
/* Heating off, or controller doesn't heat 100% -> Alarm Off*/
		if (LCPWM_DMod_var[i].x < 100)
		{
			if(i<2)
				EGM_AlarmBitField[19+i] = 0;
			else
				EGM_AlarmBitField[29+i] = 0;
		}
	}

/*Sampling der Werte für die Kurve mit einstellbarer Samplingzeit*/
	if (SamplingTime<10) SamplingTime = 100;
	Pulse.PT = SamplingTime;
	TON_10ms(&Pulse);
	if (Pulse.Q)
	{
/* take curve for showing on screen*/
		if ( TriggerLoggingOld!=TriggerLogging )
			ValueCount = 0;
		TriggerLoggingOld = TriggerLogging;
		if (TriggerLogging)
		{
/*erstes Mal? Kurve löschen*/
			if (ValueCount == 0)
			{
				int j;
				for (j=0;j<302;j++)
#ifndef TESTCURVE
				{
					Values[j] = 0;
					AmbientValues[j] = 0;
				}
#else
				{
					LCCurveByPoints_var.x = 20*j ;
					LCCurveByPoints_var2.x = 20*j;
					LCCurveByPoints(&LCCurveByPoints_var);
					LCCurveByPoints(&LCCurveByPoints_var2);
					Values[j] = EGMPreheatParam.RatedTemp[0] + LCCurveByPoints_var.y - LCCurveByPoints_var2.y;
					AmbientValues[j] = j;
				}
#endif
			}
#ifndef TESTCURVE
			Values[ValueCount] = EGMPreheat.RealTemp[0];
			AmbientValues[ValueCount] = EGMPreheat.AmbientTemp[0];
#endif
			ValueCount++;
			if(ValueCount>301)
			{
				ValueCount = 0;
				TriggerLogging = 0;
			}
			RedrawCurve = 1;
		}
		Pulse.IN = 0;
	}
	else
		Pulse.IN = 1;

/* Fester Pulstimer mit 1 sec Takt*/
	PulseTimer1.IN = 1;
	if(PulseTimer1.Q)
		PulseTimer1.IN = 0;
	TON_10ms(&PulseTimer1);

	if (PulseTimer1.Q)
	{
/*check, deviation was smaller than allowed max deviation during one minute*/
		if(RangeCheckCount>=NUMBER_OF_RANGECHECK_SECONDS)
			RangeCheckCount = 0;

		for (k=0;k<ActualNumberOfControllers;k++)
		{
			RangeCheckArray[k][RangeCheckCount] = EGMPreheat.RealTemp[k];
			EGMPreheatParam.MaxOKTemp = EGMPreheatParam.RatedTempCorr[k] + EGMPreheatParam.ToleratedDevPos;
			EGMPreheatParam.MinOKTemp = EGMPreheatParam.RatedTempCorr[k] - EGMPreheatParam.ToleratedDevNeg;
			flag[k] = TRUE;
			for (j=0;j<NUMBER_OF_RANGECHECK_SECONDS;j++)
			{
				if (	(RangeCheckArray[k][j] > EGMPreheatParam.MaxOKTemp)
				||		(RangeCheckArray[k][j] < EGMPreheatParam.MinOKTemp)	)
				{
						flag[k] = FALSE;
						break;
				}
			}
			if(ActualNumberOfControllers == 2)
				EGMPreheat.TempInRange = flag[0] && flag[1];
			else
				EGMPreheat.TempInRange = flag[0] && flag[1] && flag[2] && flag[3];

			EGMPreheat.TempNotInRange = !EGMPreheat.TempInRange;
		}
		RangeCheckCount++;
/* Alarme */
		if (ModulStatus_AT == 1)
		{

		/*Sensor defekt*/
			EGM_AlarmBitField[15] =	(EGMPreheat.RealTemp[0] > 32000 ) || (EGMPreheat.RealTemp[0] < -500 );
			EGM_AlarmBitField[16] =	(EGMPreheat.RealTemp[1] > 32000 ) || (EGMPreheat.RealTemp[1] < -500 );

			if(ActualNumberOfControllers == 4)
			{
				EGM_AlarmBitField[47] =	(EGMPreheat.RealTemp[2] > 32000 ) || (EGMPreheat.RealTemp[2] < -500 );
				EGM_AlarmBitField[48] =	(EGMPreheat.RealTemp[3] > 32000 ) || (EGMPreheat.RealTemp[3] < -500 );

				EGM_AlarmBitField[41] =	(EGMPreheat.RealTemp[2] < (EGMPreheatParam.RatedTempCorr[2] - EGMPreheatParam.ToleratedDevNeg))
								&& !EGM_AlarmBitField[47];
				EGM_AlarmBitField[42] =	(EGMPreheat.RealTemp[2] > (EGMPreheatParam.RatedTempCorr[2] + EGMPreheatParam.ToleratedDevPos))
								&& !EGM_AlarmBitField[47];

				EGM_AlarmBitField[43] =	(EGMPreheat.RealTemp[3] < (EGMPreheatParam.RatedTempCorr[3] - EGMPreheatParam.ToleratedDevNeg))
								&& !EGM_AlarmBitField[48];
				EGM_AlarmBitField[44] =	(EGMPreheat.RealTemp[3] > (EGMPreheatParam.RatedTempCorr[3] + EGMPreheatParam.ToleratedDevPos))
								&& !EGM_AlarmBitField[48];

				EGM_AlarmBitField[45] = (EGMPreheat.RealTemp[2] > (EGMPreheatParam.RatedTempCorr[2]+OVERHEATTEMP)) && !EGM_AlarmBitField[47];
				EGM_AlarmBitField[46] = (EGMPreheat.RealTemp[3] > (EGMPreheatParam.RatedTempCorr[3]+OVERHEATTEMP)) && !EGM_AlarmBitField[48];
			}
			else
			{
				EGM_AlarmBitField[41] =	0;
				EGM_AlarmBitField[42] =	0;
				EGM_AlarmBitField[43] =	0;
				EGM_AlarmBitField[44] =	0;
				EGM_AlarmBitField[45] =	0;
				EGM_AlarmBitField[46] =	0;
				EGM_AlarmBitField[47] =	0;
				EGM_AlarmBitField[48] =	0;
			}

			EGM_AlarmBitField[17] =	(EGMPreheat.AmbientTemp[0] > 32000 ) || (EGMPreheat.AmbientTemp[0] < -500 );
		/*Temp. nicht im Range*/
			EGM_AlarmBitField[8] =	(EGMPreheat.RealTemp[0] < (EGMPreheatParam.RatedTempCorr[0] - EGMPreheatParam.ToleratedDevNeg))
								&& !EGM_AlarmBitField[15];
			EGM_AlarmBitField[9] =	(EGMPreheat.RealTemp[0] > (EGMPreheatParam.RatedTempCorr[0] + EGMPreheatParam.ToleratedDevPos))
								&& !EGM_AlarmBitField[15];
			EGM_AlarmBitField[10] =	(EGMPreheat.RealTemp[1] < (EGMPreheatParam.RatedTempCorr[1] - EGMPreheatParam.ToleratedDevNeg))
								&& !EGM_AlarmBitField[16];
			EGM_AlarmBitField[11] =	(EGMPreheat.RealTemp[1] > (EGMPreheatParam.RatedTempCorr[1] + EGMPreheatParam.ToleratedDevPos))
								&& !EGM_AlarmBitField[16];
		/* Überhitzt*/
			EGM_AlarmBitField[24] = (EGMPreheat.RealTemp[0] > (EGMPreheatParam.RatedTempCorr[0]+OVERHEATTEMP)) && !EGM_AlarmBitField[15];
			EGM_AlarmBitField[25] = (EGMPreheat.RealTemp[1] > (EGMPreheatParam.RatedTempCorr[1]+OVERHEATTEMP)) && !EGM_AlarmBitField[16];
		}
		else	/* Modulsttatus nicht OK? Werte nicht gültig, also keine Fehlermeldung */
		{
			EGM_AlarmBitField[15] =	0;
			EGM_AlarmBitField[16] =	0;
			EGM_AlarmBitField[17] =	0;
			EGM_AlarmBitField[8] =	0;
			EGM_AlarmBitField[9] =	0;
			EGM_AlarmBitField[10] =	0;
			EGM_AlarmBitField[24] =	0;
			EGM_AlarmBitField[25] =	0;

			EGM_AlarmBitField[41] =	0;
			EGM_AlarmBitField[42] =	0;
			EGM_AlarmBitField[43] =	0;
			EGM_AlarmBitField[44] =	0;
			EGM_AlarmBitField[45] =	0;
			EGM_AlarmBitField[46] =	0;
			EGM_AlarmBitField[47] =	0;
			EGM_AlarmBitField[48] =	0;
		}

/* Zeitmessung f Sollwertnachführung*/
		if(SPTrackCount>NUMBER_OF_SECONDS )
			StopSPTracking = 1;

		if(ActualNumberOfControllers == 2)
		{
			if (EGMPreheat.Auto[0]
			 && EGMPreheat.Auto[1]
			 && EGMPreheat.TempInRange)
				SPTrackCount++;
		}
		else
		{
			if (EGMPreheat.Auto[0]
			 && EGMPreheat.Auto[1]
			 && EGMPreheat.Auto[2]
			 && EGMPreheat.Auto[3]
			 && EGMPreheat.TempInRange)
				SPTrackCount++;
		}
	}

/*Wert f Sollwertnachführung bestimmen (Ausgang wird in der Schleife verarbeitet)*/
	LCCurveByPoints_var.x = SPTrackCount ;
	LCCurveByPoints_var2.x = SPTrackCount ;
	LCCurveByPoints(&LCCurveByPoints_var);
	LCCurveByPoints(&LCCurveByPoints_var2);

/*********************************************************************************************/
/*********************************************************************************************/
	if (PreheatParamEnter)
	{
		PreheatParamEnter = 0;
		for (i = 0;i<ActualNumberOfControllers;i++)
		{
			LCPIDpara_var[i].enter = 1;
			LCPIDpara_var[i].Kp = EGMPreheatParam.ReglerParam[i].Kp;
			LCPIDpara_var[i].Tn = EGMPreheatParam.ReglerParam[i].Tn;
			LCPIDpara_var[i].Tv = EGMPreheatParam.ReglerParam[i].Tv;
			LCPIDpara_var[i].Tf = EGMPreheatParam.ReglerParam[i].Tf;
			LCPIDpara_var[i].Kw = EGMPreheatParam.ReglerParam[i].Kw;
			LCPIDpara_var[i].Kfbk = EGMPreheatParam.ReglerParam[i].Kfbk;
/*
			LCPWM_DMod_var[i].tminpuls = EGMPreheatParam.ReglerParam[i].tminpuls;
			LCPWM_DMod_var[i].tperiod = EGMPreheatParam.ReglerParam[i].tperiod;
*/
			LCPWM_DMod_var[i].tminpuls			= 10;  /* 10 ms kürzester Puls bzw pause*/
			LCPWM_DMod_var[i].tperiod			= 200;  /*Periodendauer 0,2 sec*/

			if ( ( EGMPreheatParam.ReglerParam[i].d_mode != LCPID_D_MODE_X )&&
				( EGMPreheatParam.ReglerParam[i].d_mode != LCPID_D_MODE_E ))
			{
				LCPIDpara_var[i].d_mode = LCPID_D_MODE_X;
				EGMPreheatParam.ReglerParam[i].d_mode = LCPID_D_MODE_X;
			}
			else
				LCPIDpara_var[i].d_mode = EGMPreheatParam.ReglerParam[i].d_mode;

		}
/*für den Fall, daß sich die Parameter geändert haben*/
		Preset_CorrCurve();
	}
	else
		for (i = 0;i<ActualNumberOfControllers;i++)
			LCPIDpara_var[i].enter = 0;

/* wenn eine der Ist-Temperaturen über ein absolutes Maximum geht ist das Preheat
überhitzt, das Overheated flag schaltet dann den Ausgang ab
*/
	if(ActualNumberOfControllers == 2)
		Overheated = (EGMPreheat.RealTemp[0] > (EGMPreheatParam.RatedTempCorr[0]+OVERHEATTEMP))
				  || (EGMPreheat.RealTemp[1] > (EGMPreheatParam.RatedTempCorr[1]+OVERHEATTEMP));
	else
		Overheated = (EGMPreheat.RealTemp[0] > (EGMPreheatParam.RatedTempCorr[0]+OVERHEATTEMP))
				  || (EGMPreheat.RealTemp[1] > (EGMPreheatParam.RatedTempCorr[1]+OVERHEATTEMP))
				  || (EGMPreheat.RealTemp[2] > (EGMPreheatParam.RatedTempCorr[2]+OVERHEATTEMP))
				  || (EGMPreheat.RealTemp[3] > (EGMPreheatParam.RatedTempCorr[3]+OVERHEATTEMP));

	if(Overheated && ControlVoltageOk)
	{
/* Not Aus erzeugen */
		ActivateControlVoltage = OFF;
		ShowMessage(136,137,0,CAUTION,OKONLY, FALSE);
	}

/*********************************************************************************************/
/* Schleife über die implementierten Regelkreise*/
/*********************************************************************************************/
	for (i = 0;i<ActualNumberOfControllers;i++)
	{
/* Parameter ungültig? dann Standard setzen*/
		if ( ( LCPIDpara_var[i].d_mode != LCPID_D_MODE_X )&&
			( LCPIDpara_var[i].d_mode != LCPID_D_MODE_E ))
		{
			LCPIDpara_var[i].d_mode	= LCPID_D_MODE_X;
			EGMPreheatParam.ReglerParam[i].d_mode = LCPID_D_MODE_X;
		}

	/*********************************************************************************************/
	/* Stellgröße auf PWM Modul geben */
		if (ControlVoltageOk && EGMPreheat.FansOn && EGMPreheat.Enable && !Overheated)
			LCPWM_DMod_var[i].x 				= LCPID_var[i].Y;
		else
			LCPWM_DMod_var[i].x 				= 0;
	/* Abtast Takt*/
		LCPWM_DMod_var[i].basetime		= LCCountVar.mscnt;

	/*  PWM Ansteuerung des Ausgangs */
		LCPWM_DMod(&LCPWM_DMod_var[i]);
		HeatingON[i] = LCPWM_DMod_var[i].y
						&& ControlVoltageOk
						&& EGMPreheat.FansOn
						&& EGMPreheat.Enable
						&& !Overheated;

	/*********************************************************************************************/
	/*********************************************************************************************/
	/*********************************************************************************************/
	/* Parametrierbaustein*/

		LCPIDpara(&LCPIDpara_var[i]);
	/*********************************************************************************************/
	/*********************************************************************************************/
	/*********************************************************************************************/
	/* AutoTune Baustein*/

	/*
	Anforderung für Autotuning
	LCPIDAUTOTUNE_REQU_OFF: Autotuning inaktiv, Regler ist freigegeben.
	LCPIDAUTOTUNE_REQU_STEPRESPONSE: Autotuning nur des Führungsverhaltens (Aufnahme einer Sprungantwort).
	LCPIDAUTOTUNE_REQU_OSCILLATE: Autotuning des Störverhaltens durch Anregen der Strecke zum Schwingen.
	LCPIDAUTOTUNE_REQU_AUTOTUNE: Autotuning des Führungsverhaltens mit anschließendem Autotuning des Störverhaltens
	*/
		if (StartAutoTune)
			LCPIDAutoTune_var[0].request				= LCPIDAUTOTUNE_REQU_AUTOTUNE;
		else
			LCPIDAutoTune_var[i].request				= LCPIDAUTOTUNE_REQU_OFF;

		LCPIDAutoTune_var[i].basetime				= LCCountVar.mscnt;

/*		LCPIDAutoTune(&LCPIDAutoTune_var[i]);*/

	/*********************************************************************************************/
	/*********************************************************************************************/
	/*********************************************************************************************/
	/* Reglerbaustein LCPID*/
	/* OHNE AUTOTUNE*/
		if( i!=0 )
			LCPID_var[i].ident						= LCPIDpara_var[i].ident;

	/* Mit AUTOTUNE*/
		if (StartAutoTune)
			LCPID_var[0].ident						= LCPIDAutoTune_var[0].ident;
		else
			LCPID_var[0].ident						= LCPIDpara_var[0].ident;

/*Sollwert tracking mit e-funktion*/
/*
		if (EGMPreheatParam.ReglerParam[i].SetpointTracking && !StopSPTracking)
			EGMPreheatParam.RatedTempCorr[i]  = EGMPreheatParam.RatedTemp[i] + LCCurveByPoints_var.y;
		else
			EGMPreheatParam.RatedTempCorr[i]  = EGMPreheatParam.RatedTemp[i];
*/
/* ENDE Sollwert tracking mit e-funktion*/

/*Sollwert tracking mit gerade f(T[ambient])*/
		if (EGMPreheatParam.ReglerParam[i].SetpointTracking )
		{
			REAL m,b;
			int CorrValue;
/* gerade wird durch 2 Punkte gelegt
x1 = EGMPreheatParam.StartAmbient[0]
y1 = (EGMPreheatParam.EndSetpoint[0] + EGMPreheatParam.StartOverheat[0])

x2 = EGMPreheatParam.StartAmbient[0]
y2 = EGMPreheatParam.EndAmbient[0]
*/

/*
	m = (y2-y1)/(x2-x1)
	b  =  y2 - m*x2  ODER  b  =  y1- m*x1
*/
			EGMPreheatParam.EndSetpoint[0] = EGMPreheatParam.RatedTemp[0];

			m = ((REAL)EGMPreheatParam.EndSetpoint[0] - (REAL)(EGMPreheatParam.EndSetpoint[0] + EGMPreheatParam.StartOverheat[0]))
				/ ((REAL)EGMPreheatParam.EndAmbient[0] - (REAL)EGMPreheatParam.StartAmbient[0]);
			b = (REAL)EGMPreheatParam.EndSetpoint[0] - m*EGMPreheatParam.EndAmbient[0];
			CorrValue =10*((m * ((REAL)EGMPreheat.AmbientTemp[0]/10.0) + (b/10.0)))
													-	EGMPreheatParam.RatedTemp[0]
													+	EGMPreheatParam.RatedTemp[i];;
			if (EGMPreheat.AmbientTemp[0] < 250)
				EGMPreheatParam.RatedTempCorr[i] = EGMPreheatParam.RatedTemp[i] + EGMPreheatParam.StartOverheat[0];
			else
/* wenn Korrigierter Wert kleiner wäre als Sollwert
dann direkt auf festen Sollwert schalten,
sonst auf korrigierten Sollwert
*/
			if ( (CorrValue < EGMPreheatParam.RatedTemp[i]) )
				EGMPreheatParam.RatedTempCorr[i] = EGMPreheatParam.RatedTemp[i];
			else
				EGMPreheatParam.RatedTempCorr[i]  = CorrValue;
		}
		else /* kein Setpoint Tracking aktiviert */
			EGMPreheatParam.RatedTempCorr[i]  = EGMPreheatParam.RatedTemp[i];
/*ENDE Sollwert tracking mit f(T[ambient])*/

		LCPID_var[i].W							= EGMPreheatParam.RatedTempCorr[i];

	/*Istwert*/
		LCPID_var[i].X							= EGMPreheat.RealTemp[i];
	/*rückgeführte Stellgröße*/
		LCPID_var[i].Y_fbk					= LCPID_var[i].Y;
	/*
	Reglerbetriebsart:
	LCPID_OUT_MODE_AUTO: Automatikbetrieb

	LCPID_OUT_MODE_MAN: Handbetrieb, Stellgröße fährt auf Y_man.
	LCPID_OUT_MODE_OPEN: Stellgröße fährt auf Y_max.
	LCPID_OUT_MODE_CLOSE: Stellgröße fährt auf Y_min.
	LCPID_OUT_MODE_FREEZE: Stellgröße wird eingefroren.

	Beim Zurückschalten aus diesen Modi auf OUT_MODE_AUTO wird eine evtl. bestehende
	Regelabweichung durch den P-Anteil ausgeregelt.

	LCPID_MODE_xxxx_JOLTFREE: Das Zurückschalten auf OUT_MODE_AUTO erfolgt völlig stoßfrei
	sofern der I-Anteil aktiviert ist!) - eine dann bestehende Regelabweichung kann aber nur sukzessiv durch den I-Anteil ausgeregelt */
		if (EGMPreheat.Auto[i])
			LCPID_var[i].out_mode				= LCPID_OUT_MODE_AUTO;
		else
			LCPID_var[i].out_mode				= LCPID_OUT_MODE_MAN;

		LCPID_var[i].basetime					= LCCountVar.mscnt;
		LCPID(&LCPID_var[i]);

/*
		if(StartAutoTune)
		{
			ReglerParam = LCPIDAutoTune_var[0].processPar;
			LCPIDpara_var[i].Kp				= ReglerParam.Kp;
			LCPIDpara_var[i].Tn				= ReglerParam.Tn;
			LCPIDpara_var[i].Tv				= ReglerParam.Tv;
			LCPIDpara_var[i].Tf				= ReglerParam.Tv/10;
		}
*/
	}/* ENDE der for-schleife über die Regler*/

}
```

- auxfunc.h (reference to Logical/GlobalIncludes/auxfunc.h)

### Program Logical/Processor/devtank (ANSIC, version 0.00.0)

#### developertank.c
```c
#ifdef _DEFAULT_INCLUDES
	#include <AsDefault.h>
#endif
/*************************************************************************************************
 Handling of Developertank

 - Heating, cooling, Temperature Measurement
 - filling, circulation, regeneration

*************************************************************************************************/
/*
#define TESTCURVE
*/
/**/
#undef TESTCURVE
/**/

#define OVERHEATTEMP 500	/* 50 °C */
#include "glob_var.h"
#include "egmglob_var.h"
#include "auxfunc.h"
#include <math.h>

extern void Replenish(void);
extern void InitRepl(void);
extern void TopUp(void);
extern void InitTopUp(void);
extern void InitProV(void);
extern void ProV(void);

TON_10ms_typ	MinOnTimeCooling;

TON_10ms_typ DeveloperLevelOKTimer,DeveloperLevelNOTOKTimer,DeveloperLevelErrorTimer,
			 CirculationPumpStartTimer,CircFlowDelay,CirculationPumpOffTimer;

TON_10ms_typ StandbyReplenishmentTimer;
TON_10ms_typ	RefillSafetyTimer,
				ReplSafetyTimer;

R_TRIGtyp	LevelOKR,LevelNOTOKR;

BOOL 	DevOldAuto;

/*um Heizkurve aufzunehmen*/
_LOCAL	BOOL	TriggerLogging,TriggerLoggingOld;
_GLOBAL int	DeveloperValues[350];
_GLOBAL	UINT	DeveloperSamplingTime;
_GLOBAL BOOL RedrawCurve,DeveloperTankParamEnter;
TON_10ms_typ	PulseTimer1;
int ValueCount;

_LOCAL	LCPWM_DMod_typ		LCPWM_DMod_var;
_LOCAL	LCPIDpara_typ			LCPIDpara_var;
_LOCAL	LCPID_typ				LCPID_var;
_LOCAL	LCPIDAutoTune_typ		LCPIDAutoTune_var;
_LOCAL	LCMovAvFilter_typ		LCMovAvFilter_var;

_LOCAL	BOOL 	StartAutoTune;
_LOCAL UINT	TopUpPumpTime;
		UINT	TopUpTmpPumpTime;

_LOCAL	BOOL	ResetOverallValues;
BOOL	DeveloperRefillActive;
BOOL	Overheated;
_LOCAL INT	TempSensorValue;
REAL tmpval;

TON_10ms_typ	PulseTimer1,SamplingTimer1;
BOOL	Pulse_1s;

void DeveloperPID_DefaultParam(void)
{
	DeveloperTankParamEnter = 0;
	DeveloperRefillActive = 0;

	LCPWM_DMod_var.tminpuls			= 1;  /* 100 ms kürzester Puls bzw pause*/
	LCPWM_DMod_var.tperiod			= 20;  /*Periodendauer 2 sec*/
	LCPWM_DMod_var.enable			= 1;
	LCPWM_DMod_var.max_value	= 100;
	LCPWM_DMod_var.min_value		= 0;

/*Sollwertabschwächung (1=AUS)*/
	LCPIDpara_var.Kw						= 1;
/*windup Dämpfung: 0=AUS*/
	LCPIDpara_var.Kfbk						= 0;
	LCPIDpara_var.enable					= 1;
	LCPIDpara_var.Y_max				= 100;
	LCPIDpara_var.Y_min					= -100;
	LCPIDpara_var.dY_max				= 0; /* 0= keine Rampe*/
	/*
	Rückführmodus der Stellgröße
	LCPID_FBK_MODE_INTERN: intern
	LCPID_FBK_MODE_EXTERN: extern für Ablöseregelung
	LCPID_FBK_MODE_EXT_SELECTOR: extern für Selektorregelung. In diesem Modus wird der I-Anteil des momentan nicht selektierten Reglers (Y_fbk ? Y) nach der
	Formel Yi = Y_fbk – Yp – Yd – A dem Eingang Y_fbk nachgeführt.
	*/
	LCPIDpara_var.fbk_mode				= LCPID_FBK_MODE_INTERN;
	/*
	Differenziermodus
	LCPID_D_MODE_X: nur -X (Istwert)
	LCPID_D_MODE_E: e (Regelabweichung, wie bei einem Standard- PID- Regler )
	*/
	LCPIDpara_var.d_mode				= LCPID_D_MODE_X;
	/*
	Rechenmodus:
	LCPID_CALC_MODE_EXACT: Genau (Alle Berechnungen erfolgen in Double Float - keine Rundungsfehler, auf SG3-Zentraleinheiten lange Rechenzeiten).
	LCPID_CALC_MODE_FAST: Schnell (Alle Berechnungen erfolgen in Integer - es kann zu geringfügigen Rundungsfehlern kommen, wird auch auf SG3-Zentraleinheiten sehr schnell gerechnet)
	*/
	LCPIDpara_var.calc_mode			= LCPID_CALC_MODE_EXACT;

/* Reglerbaustein LCPID*/
	LCPID_var.enable					= 1;
/*Stellgröße Handbetrieb */
	LCPID_var.Y_man					= 0;
	/*Aufschaltgröße*/
	LCPID_var.A							= 0;
	/*I-Anteil einfrieren*/
	LCPID_var.hold_I					= 0;

/* Autotune*/
	LCPIDAutoTune_var.enable				= 1;
	LCPIDAutoTune_var.Y_max				= 100;
	LCPIDAutoTune_var.Y_min				= 0;
	LCPIDAutoTune_var.P_manualAdjust		= 0;
	LCPIDAutoTune_var.I_manualAdjust		= 0;
	LCPIDAutoTune_var.D_manualAdjust		= 0;
	StartAutoTune = 0;

}

_INIT void init()
{
/*sinnvolle defaultwerte*/
	EGMDeveloperTankParam.ToleratedDevPos = 50;
	EGMDeveloperTankParam.ToleratedDevNeg = 50;
	DeveloperSamplingTime = 3000;
	TriggerLogging = 0;
	ValueCount = 0;
	DeveloperPID_DefaultParam();
	StandbyReplenishmentTimer.IN = 0;
	StandbyReplenishmentTimer.PT = 360000; /* 1 h */
	ResetOverallValues = 0;
	ReplenisherCounter = 0;
	LCMovAvFilter_var.enable 	= TRUE;
	LCMovAvFilter_var.x			= 0;
	LCMovAvFilter_var.base		= 128;
	LCMovAvFilter(&LCMovAvFilter_var);
	PulseTimer1.IN = 0;
	PulseTimer1.PT = 100;
	DeveloperLevelOKTimer.IN = 0;
	DeveloperLevelNOTOKTimer.IN = 0;
	DeveloperLevelErrorTimer.IN = 0;
	InitRepl();
	InitTopUp();
	InitProV();
}

_CYCLIC void cyclic()
{
	PulseTimer1.IN = 1;
	if(PulseTimer1.Q)
		PulseTimer1.IN = 0;
	TON_10ms(&PulseTimer1);
	Pulse_1s = PulseTimer1.Q;

/* Korrekturwert für Entwicklertemperatur verwenden*/
	EGMDeveloperTank.RealTemp = TempSensorValue + EGMDeveloperTankParam.TempOffset;
/*  Pulstimer mit 30 sec Takt*/
	SamplingTimer1.IN = 1;
	SamplingTimer1.PT = DeveloperSamplingTime;
	if(SamplingTimer1.Q)
		SamplingTimer1.IN = 0;
	TON_10ms(&SamplingTimer1);

	if (SamplingTimer1.Q)
	{
/* take curve for showing on screen*/
		if ( TriggerLoggingOld!=TriggerLogging )
			ValueCount = 0;
		TriggerLoggingOld = TriggerLogging;
		if (TriggerLogging)
		{
/*erstes Mal? Kurve löschen*/
			if (ValueCount == 0)
			{
				int j;
				for (j=0;j<302;j++)
#ifndef TESTCURVE
					DeveloperValues[j] = 0;
#else
/*TEST ONLY*/
				{
					DeveloperValues[j] = EGMDeveloperTankParam.RatedTemp + j/10;
				}
#endif
			}
#ifndef TESTCURVE
			DeveloperValues[ValueCount] = EGMDeveloperTank.RealTemp;
#endif

			ValueCount++;
			if(ValueCount>301)
			{
				ValueCount = 0;
				TriggerLogging = 0;
			}
			RedrawCurve = 1;
		}
	}

	if (DeveloperTankParamEnter)
	{
		DeveloperTankParamEnter = 0;
		LCPIDpara_var.enter = 1;
		LCPIDpara_var.Kp = EGMDeveloperTankParam.ReglerParam.Kp;
		LCPIDpara_var.Tn = EGMDeveloperTankParam.ReglerParam.Tn;
		LCPIDpara_var.Tv = EGMDeveloperTankParam.ReglerParam.Tv;
		LCPIDpara_var.Tf = EGMDeveloperTankParam.ReglerParam.Tf;
		LCPIDpara_var.Kw = EGMDeveloperTankParam.ReglerParam.Kw;
		LCPIDpara_var.Kfbk = EGMDeveloperTankParam.ReglerParam.Kfbk;
/*
		LCPWM_DMod_var.tminpuls = EGMDeveloperTankParam.ReglerParam.tminpuls;
		LCPWM_DMod_var.tperiod = EGMDeveloperTankParam.ReglerParam.tperiod;
*/
		LCPWM_DMod_var.tminpuls			= 1;  /* 100 ms kürzester Puls bzw pause*/
		LCPWM_DMod_var.tperiod			= 20;  /*Periodendauer 2 sec*/
		if ( ( EGMDeveloperTankParam.ReglerParam.d_mode != LCPID_D_MODE_X )&&
			( EGMDeveloperTankParam.ReglerParam.d_mode != LCPID_D_MODE_E ))
		{
			LCPIDpara_var.d_mode = LCPID_D_MODE_X;
			EGMDeveloperTankParam.ReglerParam.d_mode = LCPID_D_MODE_X;
		}
		else
			LCPIDpara_var.d_mode = EGMDeveloperTankParam.ReglerParam.d_mode;

	}
	else
		LCPIDpara_var.enter = 0;

/***************************************************************/
/***************************************************************/
/***************************************************************/
/***************************************************************/
/* Parameter ungültig? dann Standard setzen*/
	if ( ( LCPIDpara_var.d_mode != LCPID_D_MODE_X )&&
		( LCPIDpara_var.d_mode != LCPID_D_MODE_E ))
	{
		LCPIDpara_var.d_mode	= LCPID_D_MODE_X;
		EGMDeveloperTankParam.ReglerParam.d_mode = LCPID_D_MODE_X;
	}

/*********************************************************************************************/
/* Alarme */
		if (ModulStatus_AT == 1)
		{
			/*Sensor defekt*/
			EGM_AlarmBitField[18] =	 (EGMDeveloperTank.RealTemp > 32000 ) || (EGMDeveloperTank.RealTemp < -500 );
			/*Temp. nicht im Range*/
			EGM_AlarmBitField[6] = (EGMDeveloperTank.RealTemp < (INT)(EGMDeveloperTankParam.RatedTemp - EGMDeveloperTankParam.ToleratedDevNeg))
									&& !EGM_AlarmBitField[18];
			EGM_AlarmBitField[7] =	(EGMDeveloperTank.RealTemp > (INT)(EGMDeveloperTankParam.RatedTemp + EGMDeveloperTankParam.ToleratedDevPos))
									&& !EGM_AlarmBitField[18];
			/* Überhitzt*/
			EGM_AlarmBitField[26] = (EGMDeveloperTank.RealTemp > OVERHEATTEMP) && !EGM_AlarmBitField[18];
		}
		else /* Modulsttatus nicht OK? Werte nicht gültig, also keine Fehlermeldung */
		{
			EGM_AlarmBitField[18] = 0;
			EGM_AlarmBitField[6]  = 0;
			EGM_AlarmBitField[7]  = 0;
			EGM_AlarmBitField[26] = 0;
		}
/*********************************************************************************************/
/* PWM Ansteuerung des Ausgangs */
/* VAR_INPUT (analogous) */

/**
wenn alle Randbedingunge erfüllt sind, dann die Stellgröße auf den PWM Baustein geben
**/
	if (EGMDeveloperTank.LevelInRange && (EGMDeveloperTank.CoolingOn == OFF)
	&& EGMDeveloperTank.Enable
	&& !Overheated)
	{
/* solange wir mehr als 0,3 °C unterhalb sollwert sind: vollgas (Aufheizphase)
danach Regleraktivieren*/
		if(EGMDeveloperTank.RealTemp < (EGMDeveloperTankParam.RatedTemp -3))
			LCPWM_DMod_var.x 				= 100;
		else
			LCPWM_DMod_var.x 				= LCPID_var.Y;

	}
	else
		LCPWM_DMod_var.x 				= 0;

	LCPWM_DMod_var.basetime		= LCCountVar.ms100cnt;

/*  PWM Ansteuerung des Ausgangs */
	LCPWM_DMod(&LCPWM_DMod_var);

/*******************************************************************************/
/*******************************************************************************/
/* Thermo Kühl-/Heizgerät als Stellglied*/
/*******************************************************************************/
/*******************************************************************************/
/*
 * Variante Thermo Kühl/Heiz Gerät
 * Sollwert wird gemappt auf Temperaturbereich des Gerätes
 * -100% bis +100% wird zu (z.B.) 2°C bis 80°C
 * f(x) = (39/100)x + SW
 *
 * Änderung: Stellgröße beschränkt auf 10 bis 45 °C, mehr wird vom Kühlgerät
 * sowieso nicht erreicht (als Istwert)
 * f(x) = (35/200)x + SW
 */
/*
 * Filterung der Stellgröße
 */
	LCMovAvFilter_var.enable 	= TRUE;
	LCMovAvFilter_var.x			= LCPID_var.Y;

	LCMovAvFilter(&LCMovAvFilter_var);

 	tmpval = (35.0/200.0)*LCMovAvFilter_var.y + (EGMDeveloperTankParam.RatedTemp / 10.0);
	if ((LCPID_var.Y >= 100) || (tmpval > 45.0))
		Cooler.NewValues.SetPoint = 45.0;
	else
	if ((LCPID_var.Y <= -100) || (tmpval < 10.0))
		Cooler.NewValues.SetPoint = 10.0;
	else
		Cooler.NewValues.SetPoint = tmpval;

/*******************************************************************************/
/*******************************************************************************/

/* Ausgang nur ansteuern wenn Füllstand OK und Kühlung aus, sowie
Regler EIN und keine Überhitzung,
 sonst Heizung AUS*/
	EGMDeveloperTank.HeatingOn = LCPWM_DMod_var.y;

	if ((LCPWM_DMod_var.x < EGMDeveloperTankParam.CoolingOnY)
	&& EGMDeveloperTank.Enable)
		EGMDeveloperTank.CoolingOn = ON;
	else
	if (MinOnTimeCooling.Q)
		EGMDeveloperTank.CoolingOn = OFF;

	MinOnTimeCooling.PT = EGMDeveloperTankParam.MinOnTimeCooling;
	MinOnTimeCooling.IN = EGMDeveloperTank.CoolingOn;
	TON_10ms(&MinOnTimeCooling);

/*********************************************************************************************/
/*********************************************************************************************/
/*********************************************************************************************/
/* Parametrierbaustein*/

	LCPIDpara(&LCPIDpara_var);
/*********************************************************************************************/
/*********************************************************************************************/
/*********************************************************************************************/
/* AutoTune Baustein*/

/*
Anforderung für Autotuning
LCPIDAUTOTUNE_REQU_OFF: Autotuning inaktiv, Regler ist freigegeben.
LCPIDAUTOTUNE_REQU_STEPRESPONSE: Autotuning nur des Führungsverhaltens (Aufnahme einer Sprungantwort).
LCPIDAUTOTUNE_REQU_OSCILLATE: Autotuning des Störverhaltens durch Anregen der Strecke zum Schwingen.
LCPIDAUTOTUNE_REQU_AUTOTUNE: Autotuning des Führungsverhaltens mit anschließendem Autotuning des Störverhaltens
*/
	if (StartAutoTune)
		LCPIDAutoTune_var.request				= LCPIDAUTOTUNE_REQU_AUTOTUNE;
	else
		LCPIDAutoTune_var.request				= LCPIDAUTOTUNE_REQU_OFF;

	LCPIDAutoTune_var.basetime				= LCCountVar.ms100cnt;

/*	LCPIDAutoTune(&LCPIDAutoTune_var);*/

/*********************************************************************************************/
/*********************************************************************************************/
/*********************************************************************************************/
/* Reglerbaustein LCPID*/
	if (StartAutoTune)
		LCPID_var.ident						= LCPIDAutoTune_var.ident;
	else
		LCPID_var.ident						= LCPIDpara_var.ident;
/*Sollwert*/
	LCPID_var.W							= EGMDeveloperTankParam.RatedTemp;

/*Istwert*/
	LCPID_var.X							= EGMDeveloperTank.RealTemp;

/*rückgeführte Stellgröße*/
	LCPID_var.Y_fbk					= LCPID_var.Y;
/*
Reglerbetriebsart:
LCPID_OUT_MODE_AUTO: Automatikbetrieb

LCPID_OUT_MODE_MAN: Handbetrieb, Stellgröße fährt auf Y_man.
LCPID_OUT_MODE_OPEN: Stellgröße fährt auf Y_max.
LCPID_OUT_MODE_CLOSE: Stellgröße fährt auf Y_min.
LCPID_OUT_MODE_FREEZE: Stellgröße wird eingefroren.

Beim Zurückschalten aus diesen Modi auf OUT_MODE_AUTO wird eine evtl. bestehende
Regelabweichung durch den P-Anteil ausgeregelt.

LCPID_MODE_xxxx_JOLTFREE: Das Zurückschalten auf OUT_MODE_AUTO erfolgt völlig stoßfrei
sofern der I-Anteil aktiviert ist!) - eine dann bestehende Regelabweichung kann aber nur sukzessiv durch den I-Anteil ausgeregelt */
	if (EGMDeveloperTank.Auto)
		LCPID_var.out_mode				= LCPID_OUT_MODE_AUTO;
	else
		LCPID_var.out_mode				= LCPID_OUT_MODE_MAN;

	LCPID_var.basetime					= LCCountVar.ms100cnt;
	LCPID(&LCPID_var);

	if(StartAutoTune)
	{
		LCPIDpara_var.Kp				= LCPIDAutoTune_var.processPar.Kp;
		LCPIDpara_var.Tn				= LCPIDAutoTune_var.processPar.Tn;
		LCPIDpara_var.Tv				= LCPIDAutoTune_var.processPar.Tv;
		LCPIDpara_var.Tf				= LCPIDAutoTune_var.processPar.Tv/10;
	}

/***************************************************************/
/***************************************************************/
/***************************************************************/
/***************************************************************/

	EGMDeveloperTankParam.MaxOKTemp = EGMDeveloperTankParam.RatedTemp + EGMDeveloperTankParam.ToleratedDevPos;
	EGMDeveloperTankParam.MinOKTemp = EGMDeveloperTankParam.RatedTemp - EGMDeveloperTankParam.ToleratedDevNeg;

/*Measurement*/

	Overheated = EGMDeveloperTank.RealTemp > OVERHEATTEMP;

	if(	(EGMDeveloperTank.RealTemp <= EGMDeveloperTankParam.MaxOKTemp) &&
		(EGMDeveloperTank.RealTemp >= EGMDeveloperTankParam.MinOKTemp)
		)
		EGMDeveloperTank.TempInRange = TRUE;
	else
		EGMDeveloperTank.TempInRange = FALSE;

	EGMDeveloperTank.TempNotInRange = !EGMDeveloperTank.TempInRange;

/*Level*/
	DeveloperLevelOKTimer.IN = EGMDeveloperTank.TankFull;
	DeveloperLevelOKTimer.PT = 500; /*5 sec*/
	TON_10ms(&DeveloperLevelOKTimer);

	DeveloperLevelNOTOKTimer.IN = !EGMDeveloperTank.TankFull;
	DeveloperLevelNOTOKTimer.PT = 500; /*5 sec*/
	TON_10ms(&DeveloperLevelNOTOKTimer);

	LevelOKR.CLK = DeveloperLevelOKTimer.Q;
	LevelNOTOKR.CLK = DeveloperLevelNOTOKTimer.Q;
	R_TRIG(&LevelOKR);
	R_TRIG(&LevelNOTOKR);
	if(LevelOKR.Q)
		EGMDeveloperTank.LevelNotInRange = FALSE;
	if(LevelNOTOKR.Q)
		EGMDeveloperTank.LevelNotInRange = TRUE;

	EGMDeveloperTank.LevelInRange = !EGMDeveloperTank.LevelNotInRange;
/* Fehlermeldung verzögern, erst wird automatisch befüllt */
	DeveloperLevelErrorTimer.IN = EGMDeveloperTank.LevelNotInRange;
	DeveloperLevelErrorTimer.PT = 2000; /* 20 s */
	TON_10ms(&DeveloperLevelErrorTimer);
	EGM_AlarmBitField[5] = (ModulStatus_DI == 1) && DeveloperLevelErrorTimer.Q;

/*auto-refill and circulation*/
	CirculationPumpOffTimer.IN = EGMDeveloperTank.LevelNotInRange;
	CirculationPumpOffTimer.PT = 2000; /*20 sec */
	TON_10ms(&CirculationPumpOffTimer);

	if(	EGMGlobalParam.UseDevCircFlowControl )
	{
		CirculationPumpStartTimer.IN = EGMDeveloperTank.CirculationPump;
		CirculationPumpStartTimer.PT = 1000; /* 10 sec */
		TON_10ms(&CirculationPumpStartTimer);
		CircFlowDelay.IN = !DevCircFlowInput;
		CircFlowDelay.PT = 300; /* 3 sec */
		TON_10ms(&CircFlowDelay);
		if( CirculationPumpStartTimer.Q && CircFlowDelay.Q )
		{
			EGM_AlarmBitField[34] = TRUE;
			EGMDeveloperTank.CirculationPump = OFF;
		}
	}
	else
		EGM_AlarmBitField[34] = FALSE;

	if (EGMDeveloperTank.Auto )
	{
		if ( CirculationPumpOffTimer.Q || EGM_AlarmBitField[34] )
			EGMDeveloperTank.CirculationPump = OFF;
		else
		if (EGMDeveloperTank.LevelInRange)
			EGMDeveloperTank.CirculationPump = ON;

		if (EGMDeveloperTank.LevelNotInRange && !EGM_AlarmBitField[38])
		{
			EGMDeveloperTank.Refill = ON;
			DeveloperRefillActive = TRUE;
		}
		else
		if(DeveloperRefillActive)
		{
			EGMDeveloperTank.Refill = OFF;
			DeveloperRefillActive = FALSE;
		}

		/*
		* Switch Cooler On
		*/
		if( !Cooler.UnitOn && !DevOldAuto )
			Cooler.Cmd_Start = TRUE;
	}

/* AUTO mode off: stop refill pump, stop circulation*/
	if ((DevOldAuto && !EGMDeveloperTank.Auto) || !ControlVoltageOk)
	{
		EGMDeveloperTank.Refill = OFF;
		DeveloperRefillActive = FALSE;
		EGMDeveloperTank.CirculationPump = OFF;
		if( Cooler.UnitOn )
			Cooler.Cmd_Stop = TRUE;
	}
	DevOldAuto = EGMDeveloperTank.Auto;

/******************************************************************************/
/******************************************************************************/
/* REPLENISHING developer*/

	if(EGMGlobalParam.PROV_KitInstalled)
		ProV();
	else
	{
		Replenish();
		TopUp();
	}

/* Saftey: pump off, after 30 sec, if Tank is full */
	RefillSafetyTimer.IN = EGMDeveloperTank.Refill && EGMDeveloperTank.TankFull;
	RefillSafetyTimer.PT = 3000;
	if(RefillSafetyTimer.Q)
		EGMDeveloperTank.Refill = OFF;

	ReplSafetyTimer.IN = EGMDeveloperTank.RegenerationPump && EGMDeveloperTank.TankFull;
	ReplSafetyTimer.PT = 3000;
	if(ReplSafetyTimer.Q)
		EGMDeveloperTank.RegenerationPump = OFF;

}
```

- auxfunc.h (reference to Logical/GlobalIncludes/auxfunc.h)

#### replenishing.c
```c
#ifdef _DEFAULT_INCLUDES
	#include <AsDefault.h>
#endif
/*
                             *******************
******************************* C SOURCE FILE *******************************
**                           *******************                           **
**                                                                         **
** project  : BlueFin                                                      **
** filename : REPLENISHING.C                                               **
** version  : 1.01                                                         **
** date     : 29.10.2007                                                   **
**                                                                         **
*****************************************************************************
** Abstract                                                                **
** ========                                                                **
** Replenishing developer automatically controlled by sqm, number of       **
** plates, or (in Standby) by time                                         **
**                                                                         **
** Copyright (c) 2007, Krause-Biagosch GmbH                                **
** All rights reserved.                                                    **
**                                                                         **
*****************************************************************************
VERSION HISTORY:
----------------
Version     : 1.00
Date        : 05.07.2007
Revised by  : Herbert Aden
Description : Original version, moved functionality from
              developertank module to here.

Version     : 1.01
Date        : 29.10.2007
Revised by  : Herbert Aden
Description : - locking of button "manual replenishing" didn't work correctly
              ->new variable LockManualReplenishment locks only the input for
                amount of replenisher
              - Button Manual Replenishment is not locked anymore, the user
                can now stop replenishing by pressing it a 2nd time

*/
#define _REPLENISHING_C_SRC

/****************************************************************************/
/**                                                                        **/
/**                           INCLUDE FILES                                **/
/**                                                                        **/
/****************************************************************************/

#include "glob_var.h"
#include "egmglob_var.h"
#include <math.h>

/****************************************************************************/
/**                                                                        **/
/**                       DEFINITIONS AND MACROS                           **/
/**                                                                        **/
/****************************************************************************/
/* NONE */

/****************************************************************************/
/**                                                                        **/
/**                      TYPEDEFS AND STRUCTURES                           **/
/**                                                                        **/
/****************************************************************************/
/* NONE */

/****************************************************************************/
/**                                                                        **/
/**                      PROTOTYPES OF LOCAL FUNCTIONS                     **/
/**                                                                        **/
/****************************************************************************/
/* NONE */

/****************************************************************************/
/**                                                                        **/
/**                      EXPORTED VARIABLES                                **/
/**                                                                        **/
/****************************************************************************/
/* NONE */

/****************************************************************************/
/**                                                                        **/
/**                           GLOBAL VARIABLES                             **/
/**                                                                        **/
/****************************************************************************/
/***
 ShutDownTime enthält den letzten Zeitstempel vor dem letzten Ausschalten
 wird im INIT in OffTime umkopiert, weil ShutDownTime ja zyklisch beschrieben wird
 OnTime wird im INIT mit der aktuellen Zeit gesetzt, damit kann man aus der
 Differenz zwischen OnTime und OffTime ermitteln, wie lange die Maschine aus war
***/
_GLOBAL   DATE_AND_TIME       OffTime;

/****************************************************************************/
/**                                                                        **/
/**                      TASK-LOCAL VARIABLES                              **/
/**                                                                        **/
/****************************************************************************/
_LOCAL    UINT                NextReplenishingIn;	/* for display*/
/* Variables for manual replenishing*/
_LOCAL    UINT                ManualReplenishment,ManualReplenishmentMinValue;
_LOCAL    BOOL                StartManualReplenishment;
_LOCAL    BOOL                LockManualReplenishment; /* to lock the button
                                                        * while replenishing
                                                        * active
                                                        */
_LOCAL    UINT                PumpTime,PumpTimeToGo;
_LOCAL    UINT                TopUpPumpTime;

/****************************************************************************/
/**                                                                        **/
/**                    MODULE-LOCAL VARIABLES                              **/
/**                                                                        **/
/****************************************************************************/
static    UINT                ReplStep,TopUpStep;
static    UDINT               StandbyReplenishmentSeconds; /*
                                                            * count seconds
                                                            * until next
                                                            * standbyrepl.
                                                            */
static    BOOL                OffReplenishingDone,ManualReplenishmentStarted;
static    REAL                ReplAmount;
static    TON_10ms_typ        ReplTimer,ReplenishmentFlowCheckTimer;
static    REAL                TopUpAmount;
static    TON_10ms_typ        TopUpTimer,TopUpFlowCheckTimer;

/****************************************************************************/
/**                                                                        **/
/**                      EXTERNAL VARIABLES                                **/
/**                                                                        **/
/****************************************************************************/
extern BOOL	Pulse_1s;

/****************************************************************************/
/**                                                                        **/
/**                          EXPORTED FUNCTIONS                            **/
/**                                                                        **/
/****************************************************************************/

void InitRepl(void)
{
	StandbyReplenishmentSeconds = 0;
	OffReplenishingDone = 0;
	ReplTimer.IN = 0;
	ReplTimer.PT = 1000;
	LockManualReplenishment = FALSE;
}

void InitTopUp(void)
{
	StandbyReplenishmentSeconds = 0;
	TopUpTimer.IN = 0;
	TopUpTimer.PT = 1000;
}

void Replenish(void)
{

	TON_10ms(&ReplTimer);

	switch (ReplStep)
	{
/*
 * Wait for condition to start replenishing
 * and calculate amount and pump running time
 */
		case 0:
		{
			ManualReplenishmentStarted = FALSE;
/* a) Standby*/
			if( EGMDeveloperTankParam.EnableStandbyReplenishing
		     && (CurrentState != S_PROCESSING)
		     )
			{
				if( Pulse_1s )
					StandbyReplenishmentSeconds++;

				if (StandbyReplenishmentSeconds >
						(EGMDeveloperTankParam.StandbyReplenishmentIntervall * 60))
				{
				/* calc. running time of pump:
				 * ((ml/h) * hours) / (ml/s)
				 */

					PumpTime =
						((EGMDeveloperTankParam.StandbyReplenishment  * ( StandbyReplenishmentSeconds/3600.0)) / EGMDeveloperTankParam.PumpMlPerSec)*100;
					if (PumpTime >= EGMDeveloperTankParam.MinPumpOnTimeStandby)
					{
						ReplAmount =
							(EGMDeveloperTankParam.StandbyReplenishment  * ( StandbyReplenishmentSeconds/3600.0));
						ReplStep = 10;
						StandbyReplenishmentSeconds = 0;
					}
					NextReplenishingIn = 0;
				}
				else	/* calc display value "next replenishinh in XX min"*/
					NextReplenishingIn = EGMDeveloperTankParam.StandbyReplenishmentIntervall -
											(StandbyReplenishmentSeconds/60.0);

			}

/**************************************************************************************/
/* OFF Replenishing, only once on startup*/
			if (EGMDeveloperTankParam.EnableOffReplenishing
				&&(!OffReplenishingDone) )
			{

				PumpTime =
						((EGMDeveloperTankParam.OffReplenishment  * ( OffTime/3600.0)) / EGMDeveloperTankParam.PumpMlPerSec)*100;
				if (PumpTime >= EGMDeveloperTankParam.MinPumpOnTimeStandby
				/*mehr als 5 l Regenerat -> da ist was faul, wir regenieren nicht*/
				&& ((EGMDeveloperTankParam.OffReplenishment  * ( OffTime/3600.0)) < 5000)
				)
				{
					ReplAmount =
						(EGMDeveloperTankParam.OffReplenishment  * ( OffTime/3600.0));
					ReplStep = 10;
				}
				OffReplenishingDone = 1;
			}

/**************************************************************************************/
/* b) per plate*/
			if (Pulse_1s &&(CurrentState == S_PROCESSING)&& (EGMDeveloperTankParam.ReplenishingMode == REPLPERPLATE))
			{
				PumpTime =
						((ReplenishmentPlateCounter * EGMDeveloperTankParam.ReplenishmentPerPlate) / EGMDeveloperTankParam.PumpMlPerSec)*100;
				if (PumpTime >= EGMDeveloperTankParam.MinPumpOnTime)
				{
					ReplAmount =
						ReplenishmentPlateCounter * EGMDeveloperTankParam.ReplenishmentPerPlate;
					ReplStep = 10;
					ReplenishmentPlateCounter = 0;
				}
			}

/**************************************************************************************/
/* c) per area*/
			if (Pulse_1s &&(CurrentState == S_PROCESSING)&& (EGMDeveloperTankParam.ReplenishingMode == REPLPERSQM))
			{
				PumpTime =
						((ReplenishmentSqmCounter * EGMDeveloperTankParam.ReplenishmentPerSqm) / EGMDeveloperTankParam.PumpMlPerSec)*100;
				if (PumpTime >= EGMDeveloperTankParam.MinPumpOnTime)
				{
					ReplAmount =
						ReplenishmentSqmCounter * EGMDeveloperTankParam.ReplenishmentPerSqm;
					ReplStep = 10;

					ReplenishmentSqmCounter = 0;
				}
			}

/**************************************************************************************/
/* d) manually*/
			ManualReplenishmentMinValue = EGMDeveloperTankParam.PumpMlPerSec * (EGMDeveloperTankParam.MinPumpOnTime/100.0);
			if (StartManualReplenishment)
			{
				PumpTime =
						(ManualReplenishment / EGMDeveloperTankParam.PumpMlPerSec)*100;
				if (PumpTime >= EGMDeveloperTankParam.MinPumpOnTime)
				{
					ReplAmount = ManualReplenishment;
					ReplStep = 10;
					ManualReplenishmentStarted = TRUE;
					LockManualReplenishment = TRUE;
				}
			}

			ReplTimer.IN = 0;
			break;
		}

/*
 * - if pump is running, wait
 * - reset flow counter if flow control is in use
 *
 */
		case 10:
		{
			if( EGMDeveloperTank.RegenerationPump == ON )
				break;
/* reset Error message */
			EGM_AlarmBitField[37] = FALSE;
			if( EGMGlobalParam.UseReplFlowControl )
			{
				ReplFC.ResetMlFlown = TRUE;
				ReplStep = 12;
			}
			else
				ReplStep = 20;

			break;
		}
/*
 * if flow control is in use, wait for counter reset
 */
		case 12:
		{
			if( ReplFC.ResetMlFlown == FALSE )
				ReplStep = 20;
			break;
		}

/*
 * - start pump
 * - start timer
 */
		case 20:
		{
			EGMDeveloperTank.RegenerationPump = ON;
			if( EGMGlobalParam.UseReplFlowControl )
				ReplTimer.PT = 6000; /* 60 sec timeout */
			else
			/* no flow control: pump is timer controlled */
				ReplTimer.PT = PumpTime;

			ReplTimer.IN = 1;
		 	ReplStep = 30;
			break;
		}

/*
 * - if flow control active, wait for amount to be flown and check for timeout
 * - else wait for timer to finish
 * - then Switch off pump
 * - calculate PumpTimeToGo
 */
		case 30:
		{
			if( !StartManualReplenishment && ManualReplenishmentStarted)
			{
				EGMDeveloperTank.RegenerationPump = OFF;
				ReplTimer.IN = 0;
				ReplStep = 40;
			}

			if( PumpTime > ReplTimer.ET )
				PumpTimeToGo = PumpTime - ReplTimer.ET;
			else
				PumpTimeToGo = 0;

			if( EGMGlobalParam.UseReplFlowControl )
			{
				if( ReplFC.MlFlown >= ReplAmount ) /* Menge erreicht */
				{
					REAL tmpval;
					if( (ReplFC.MlFlown > 0.1)
					 && (ReplTimer.ET > 0)
					 )
					 {
						tmpval = ReplFC.MlFlown / ((REAL)ReplTimer.ET / 100.0);
						if( tmpval < 1.0 )
							EGMDeveloperTankParam.PumpMlPerSec = 19.0;
						else
							EGMDeveloperTankParam.PumpMlPerSec = tmpval;
					}
					else
						EGMDeveloperTankParam.PumpMlPerSec = 20.0;

					saveParameterData = 1;
					EGMDeveloperTank.RegenerationPump = OFF;
					ReplTimer.IN = 0;
					ReplStep = 40;
					OverallReplenisherCounter += ReplFC.MlFlown;
					ReplenisherCounter += ReplFC.MlFlown;
					ReplenisherUsedSinceDevChg += ReplFC.MlFlown;
				}
				else
				/* Menge noch nicht erreicht: warten und timeout checken*/
				{
					if( (EGM_AlarmBitField[37] == TRUE) /* no flow error */
					||  ReplTimer.Q ) /* Timeout -> Error */
					{
						ReplTimer.IN = 0;
						ReplStep = 40;
						EGMDeveloperTank.RegenerationPump = OFF;
						EGM_AlarmBitField[37] = TRUE;
						ReplFC.ResetMlFlown = TRUE;
						break;
					}
					else
					/* pump switched off manually */
					if( EGMDeveloperTank.RegenerationPump == OFF )
					{
						ReplTimer.IN = 0;
						ReplStep = 40;
						break;
					}
				}
			}
			else /* no flow control */
			{
				if( ReplTimer.Q ) /* Zeit abgelaufen -> dosieren fertig */
				{
					ReplTimer.IN = 0;
					ReplStep = 40;
					EGMDeveloperTank.RegenerationPump = OFF;
					OverallReplenisherPumpTime += (ReplTimer.PT/100.0);
					OverallReplenisherCounter += ((ReplTimer.PT/100.0)* EGMDeveloperTankParam.PumpMlPerSec);
					ReplenisherCounter += ((ReplTimer.PT/100.0)* EGMDeveloperTankParam.PumpMlPerSec);
					ReplenisherUsedSinceDevChg += ((ReplTimer.PT/100.0)* EGMDeveloperTankParam.PumpMlPerSec);
				}
			}
			break;
		}

/*
 * finished: cleanup
 */
		case 40:
		{
			StartManualReplenishment = FALSE;
			LockManualReplenishment = FALSE;
			ReplTimer.IN = 0;
			ReplStep = 0;
			PumpTimeToGo = 0;
			break;
		}
	}

	if( EGMGlobalParam.UseReplFlowControl)
	{
		/* Überwachen, ob auch was kommt */
		ReplenishmentFlowCheckTimer.IN = EGMDeveloperTank.RegenerationPump;
		ReplenishmentFlowCheckTimer.PT = 1000; /* 10 sec*/
		TON_10ms(&ReplenishmentFlowCheckTimer);
		if( ReplenishmentFlowCheckTimer.Q && !ReplFC.Flowing )
		{
		/* no flow detected: stop pump and trigger error message */
			EGM_AlarmBitField[37] = TRUE;
			EGMDeveloperTank.RegenerationPump = OFF;
			StartManualReplenishment = FALSE;
		}
	}
	else /* No Flow Control */
	{
		EGM_AlarmBitField[37] = FALSE;
	} /* else */

}

/******************************************************************************/
/******************************************************************************/
/******************************************************************************/
/******************************************************************************/

void TopUp(void)
{

	TON_10ms(&TopUpTimer);

	if(isnan(EGMDeveloperTankParam.TopUpPumpMlPerSec))
	{
		EGMDeveloperTankParam.TopUpPumpMlPerSec = 20.0;
		saveParameterData = 1;
	}

	switch (TopUpStep)
	{
/*
 * Wait for condition to start topup
 * and calculate amount and pump running time
 */
		case 0:
		{

/**************************************************************************************/
/* a) per plate*/
			if (Pulse_1s &&(CurrentState == S_PROCESSING)&& (EGMDeveloperTankParam.TopUpMode == REPLPERPLATE))
			{
				TopUpPumpTime =
						((TopUpPlateCounter * EGMDeveloperTankParam.TopUpPerPlate) / EGMDeveloperTankParam.TopUpPumpMlPerSec)*100;
				if (TopUpPumpTime >= EGMDeveloperTankParam.TopUpMinPumpOnTime)
				{
					/* value for Sensorcontrolled replenishing */
					TopUpAmount =
						TopUpPlateCounter * EGMDeveloperTankParam.TopUpPerPlate;
					TopUpStep = 10;
					TopUpPlateCounter = 0;
				}
			}

/**************************************************************************************/
/* b) per area*/
			if (Pulse_1s &&(CurrentState == S_PROCESSING)&& (EGMDeveloperTankParam.TopUpMode == REPLPERSQM))
			{
				TopUpPumpTime =
						((TopUpSqmCounter * EGMDeveloperTankParam.TopUpPerSqm) / EGMDeveloperTankParam.TopUpPumpMlPerSec)*100;
				if (TopUpPumpTime >= EGMDeveloperTankParam.TopUpMinPumpOnTime)
				{
					/* value for Sensorcontrolled replenishing */
					TopUpAmount =
						TopUpSqmCounter * EGMDeveloperTankParam.TopUpPerSqm;
					TopUpStep = 10;
					TopUpSqmCounter = 0;
				}
			}

			TopUpTimer.IN = 0;
			break;
		}

/*
 * - if pump is running, wait
 * - reset flow counter if flow control is in use
 *
 */
		case 10:
		{
			if( EGMDeveloperTank.Refill == ON )
				break;
/* reset Error message */
			EGM_AlarmBitField[38] = FALSE;
			if( EGMGlobalParam.UseTopUpFlowControl )
			{
				TopUpFC.ResetMlFlown = TRUE;
				TopUpStep = 12;
			}
			else
				TopUpStep = 20;

			break;
		}
/*
 * if flow control is in use, wait for counter reset
 */
		case 12:
		{
			if( TopUpFC.ResetMlFlown == FALSE )
				TopUpStep = 20;
			break;
		}

/*
 * - start pump
 * - start timer
 */
		case 20:
		{
			EGMDeveloperTank.Refill = ON;
			if( EGMGlobalParam.UseTopUpFlowControl )
				TopUpTimer.PT = 6000; /* 60 sec timeout */
			else
			/* no flow control: pump is timer controlled */
				TopUpTimer.PT = TopUpPumpTime;

			TopUpTimer.IN = 1;
		 	TopUpStep = 30;
			break;
		}

/*
 * - if flow control active, wait for amount to be flown and check for timeout
 * - else wait for timer to finish
 * - then Switch off pump
 */
		case 30:
		{
			if( EGMGlobalParam.UseTopUpFlowControl )
			{
				if( TopUpFC.MlFlown >= TopUpAmount ) /* Menge erreicht */
				{
					REAL tmpval;
					if( (TopUpFC.MlFlown > 0.1)
					 && (TopUpTimer.ET > 0)
					 )
					 {
						tmpval = TopUpFC.MlFlown / ((REAL)TopUpTimer.ET / 100.0);
						if( tmpval < 1.0 )
							EGMDeveloperTankParam.TopUpPumpMlPerSec = 19.0;
						else
							EGMDeveloperTankParam.TopUpPumpMlPerSec = tmpval;
					}
					else
						EGMDeveloperTankParam.TopUpPumpMlPerSec = 20.0;

					saveParameterData = 1;
					EGMDeveloperTank.Refill = OFF;
					TopUpTimer.IN = 0;
					TopUpStep = 40;
				}
				else
				/* Menge noch nicht erreicht: warten und timeout checken*/
				{
					if( (EGM_AlarmBitField[38] == TRUE) /* no flow error */
					||  TopUpTimer.Q ) /* Timeout -> Error */
					{
						TopUpTimer.IN = 0;
						TopUpStep = 40;
						EGMDeveloperTank.Refill = OFF;
						EGM_AlarmBitField[38] = TRUE;
						TopUpFC.ResetMlFlown = TRUE;
						break;
					}
					else
					/* pump switched off manually */
					if( EGMDeveloperTank.Refill == OFF )
					{
						TopUpTimer.IN = 0;
						TopUpStep = 40;
						break;
					}
				}
			}
			else /* no flow control */
			{
				if( TopUpTimer.Q ) /* Zeit abgelaufen -> dosieren fertig */
				{
					TopUpTimer.IN = 0;
					TopUpStep = 40;
					EGMDeveloperTank.Refill = OFF;
				}
			}
			break;
		}

/*
 * finished: cleanup
 */
		case 40:
		{
			TopUpTimer.IN = 0;
			TopUpStep = 0;
			break;
		}
	}

	if( EGMGlobalParam.UseTopUpFlowControl)
	{
		/* Überwachen, ob auch was kommt */
		TopUpFlowCheckTimer.IN = EGMDeveloperTank.Refill;
		TopUpFlowCheckTimer.PT = 1000; /* 10 sec*/
		TON_10ms(&TopUpFlowCheckTimer);
		if( TopUpFlowCheckTimer.Q && !TopUpFC.Flowing )
		{
		/* no flow detected: stop pump and trigger error message */
			EGM_AlarmBitField[38] = TRUE;
			EGMDeveloperTank.Refill = OFF;
		}
	}
	else /* No Flow Control */
	{
		EGM_AlarmBitField[38] = FALSE;
	} /* else */

}
```
